// TwinCAT 3 PLC project SPS1
// Title: SPS PlattformCD
// Company: Gesim
// Author: U.Seifert
// ProjectVersion: 2.0.18.17
// ProgramVersion: 3.1.4022.4
// CompilerDefines: C6015, WIN10
// libraries:
//   Tc2_Math, * (Beckhoff Automation GmbH)
//   Tc2_NCI, * (Beckhoff Automation GmbH)
//   Tc2_Standard, * (Beckhoff Automation GmbH)
//   Tc2_System, * (Beckhoff Automation GmbH)
//   Tc3_Interfaces, * (Beckhoff Automation GmbH)
//   Tc3_Module, * (Beckhoff Automation GmbH)
//   Tc3_PackML, * (Beckhoff Automation GmbH)
//   Tc2_EtherCAT,newest,Beckhoff Automation GmbH
//   Tc2_IoFunctions,newest,Beckhoff Automation GmbH
//   Tc2_MC2,newest,Beckhoff Automation GmbH
//   Tc2_SerialCom,newest,Beckhoff Automation GmbH
//   Tc2_SUPS,newest,Beckhoff Automation GmbH
//   Tc2_SystemCX,newest,Beckhoff Automation GmbH
//   Tc2_Utilities,newest,Beckhoff Automation GmbH
//   Tc3_LinMot,1.0.0.3,NTI AG
//   Tc3_MemMan,newest,Beckhoff Automation GmbH
// project tree:
//   Actions/ ActionDispacher.TcPOU, FB_ActionList.TcPOU, FB_ActionStatusList.TcPOU, FB_ComplexAction.TcPOU, FB_DelayAction.TcPOU, FB_MeasTip.TcPOU, FB_MoveToTarget.TcPOU
//   / ComTask.TcTTO, GCodeTask.TcTTO, PlcTask.TcTTO
//   Configuration/ FB_Configuration.TcPOU, FB_GetObjPropChecksum.TcPOU, FB_IdPool.TcPOU, FB_ObjCollection.TcPOU, FB_ObjCollectionNode.TcPOU, FB_ObjCollectIterator.TcPOU, FB_ObjCollectIteratorDeep.TcPOU, FB_ObjectDirectory.TcPOU, GVL_ObjectArrays.TcGVL, GVL_ObjectConstants.TcGVL, GVL_ObjMgmt.TcGVL, ST_IdNode.TcDUT
//   DUTs/Enums/ E_ActionStatus.TcDUT, E_ArrayOrder.TcDUT, E_Condition.TcDUT, E_CrashAvoidanceMode.TcDUT, E_DilPrepareMode.TcDUT, E_DilPumpMode.TcDUT, E_DilType.TcDUT, E_DilValveType.TcDUT, E_DispenserState.TcDUT, E_DrivingPinCtrl.TcDUT, E_DrivingPinSelection.TcDUT, E_DrivingPinState.TcDUT, E_ErrorIdDS402.TcDUT, E_ErrorIdGCode.TcDUT, E_ErrorIdCan.TcDUT, E_ErrorIdHwGeneral.TcDUT, E_ExchangePieceOption.TcDUT, E_ExtruderType.TcDUT, E_GCodeState.TcDUT, E_GripperState.TcDUT, E_HardwarePropType.TcDUT, E_InteractMessageType.TcDUT, E_InterlockState.TcDUT, E_CompOperator.TcDUT, E_LockCtrl.TcDUT, E_LockState.TcDUT, E_MeasureMode.TcDUT, E_MeasureOption.TcDUT, E_MethodState.TcDUT, E_ModalDesignationAbsInc.TcDUT, E_ModalGeoTypes.TcDUT, E_MoveDirection.TcDUT, E_MoveMode.TcDUT, E_ObjectGroup.TcDUT, E_OpClCtrl.TcDUT, E_OpClState.TcDUT, E_LogicOperator.TcDUT, E_PickPutMode.TcDUT, E_POU.TcDUT, E_POUACT.TcDUT, E_PressCtrl.TcDUT, E_PrintParamType.TcDUT, E_ProcDataType.TcDUT, E_StackerRotPosition.TcDUT, E_SwivelCtrl.TcDUT, E_SwivelState.TcDUT, E_TargetRef.TcDUT, E_Action.TcDUT, E_ErrorIdCmd.TcDUT, E_ErrorIdDiluter.TcDUT, E_ErrorIdMultiZ.TcDUT, E_HardwareGrp.TcDUT, E_MachineMode.TcDUT, E_MachineState.TcDUT, E_ObjectType.TcDUT, E_ErrorIdObjMgmt.TcDUT, E_TeachTrgtOption.TcDUT, E_TipCleaningMode.TcDUT, E_TransferTrayCtrl.TcDUT, E_TrayHollowSelection.TcDUT, E_TriggerOutput.TcDUT, E_WashMode.TcDUT
//   DUTs/ ERRORID.TcDUT, HARDWAREGRP.TcDUT
//   DUTs/Structs/ FB_Rectangle.TcPOU, ST_Action.TcDUT, ST_ActionStatus.TcDUT, ST_2DPoint.TcDUT, ST_3DDimension.TcDUT, ST_3DPoint.TcDUT, ST_ActionData.TcDUT, ST_ActionList.TcDUT, ST_AdsAdress.TcDUT, ST_CanMasterAddress.TcDUT, ST_Circle.TcDUT, ST_EtherCATMaster.TcDUT, ST_HardwareProcData.TcDUT, ST_HardwareId.TcDUT, ST_HardwareInfo.TcDUT, ST_Interaction.TcDUT, ST_Line.TcDUT, ST_MethResult.TcDUT, ST_ObjHasMoved.TcDUT, ST_PlcInfo.TcDUT, ST_ObjectProcData.TcDUT, ST_Rectangle.TcDUT, ST_CmdData.TcDUT, ST_Error.TcDUT, ST_StepStatus.TcDUT, ST_WashPoint.TcDUT, ST_WashStep.TcDUT, ST_WasteChannel.TcDUT, ST_LiquidChannel.TcDUT, ST_RinseChannel.TcDUT
//   DUTs/Unions/ U_AdsData.TcDUT, U_ByteArr4_DINT.TcDUT, U_SDO_DATA.TcDUT
//   FirmwUpdate/ E_FirmwUpdState.TcDUT, E_S19RecordState.TcDUT, FB_S19File.TcPOU, FB_S19Record.TcPOU, FirmwUpdate.TcPOU, ST_FirmwUpdInfo.TcDUT
//   Functions/ F_Add3DPoints.TcPOU, F_CuboidInnerCuboid.TcPOU, F_GET_GCODE_NCLINE.TcPOU, F_Sub3DPoints.TcPOU, F_SynchronizeSpeeds.TcPOU
//   GCode/ E_SAF_State.TcDUT, FB_BuildGroup.TcPOU, FB_ClearGroup.TcPOU, FB_Cuboid.TcPOU, FB_FastMFunc.TcPOU, FB_HskMFunc.TcPOU, FB_RestartPrintAction.TcPOU, GCode.TcPOU, ST_GCodeInfo2.TcDUT, ST_GCodeRef.TcDUT, ST_GCodeTool.TcDUT, ST_NciInfo.TcDUT, ST_GCodeInfo.TcDUT
//   GVLs/ GVL_Hardware.TcGVL, GVL_RS232.TcGVL, GVL_Sm.TcGVL
//   Hardware/4ChannelHeater/ FB_HwRef4ChHeater.TcPOU
//   Hardware/BottleRack/ FB_HwRefBottleRack.TcPOU
//   Hardware/ CANInterfaceCom.TcPOU, E_CoDS402HomingState.TcDUT, E_CoDS402States.TcDUT, FB_CanNodeBase.TcPOU, FB_CANOpenMotionPower.TcPOU, FB_HwModule.TcPOU, FB_HwModuleList.TcPOU, FB_SendCanMessage.TcPOU, F_GetCoDS402State.TcPOU, F_CompVersion.TcPOU, HwInfoList.TcPOU, PerformHardware.TcPOU, ScanHwModules.TcPOU, SimutateHwModules.TcPOU, ST_CANInterfaceBuffer.TcDUT
//   Hardware/Diluter/ FB_Dil_GetValveConfig.TcPOU, FB_Dil_GetValvePos.TcPOU, FB_Dil_GetPlungerPos.TcPOU, FB_Dil_Pump.TcPOU, FB_Dil_MoveValve.TcPOU, FB_Dil_MoveToPos.TcPOU, FB_Dil_SendCmd.TcPOU, FB_Dil_SetValveConfig.TcPOU, FB_Dil_Transfer.TcPOU, FB_Dil_Init.TcPOU, FB_Dil_Stop.TcPOU, FB_HwRefDiluter.TcPOU, F_DilFlowToSpeed.TcPOU, F_DilQuantityToMicroSteps.TcPOU, F_GetChannelCodeTwin.TcPOU, F_GetCheckSumByte.TcPOU, F_GetCheckSumFromString.TcPOU, F_GetPumpString.TcPOU, F_GetValveCode.TcPOU
//   Hardware/EL70xxDrive/ E_EL70xx_EncoderType.TcDUT, E_EL70xx_StartType.TcDUT, FB_HWECtrl_EL70xx_Home.TcPOU, FB_HWECtrl_EL70xx_Move.TcPOU, FB_HWECtrl_EL70xx_Power.TcPOU, FB_HwRefEL70xxDrive.TcPOU, FB_HwRefEL70xxDriveExtEncoder.TcPOU, ST_EL70xx_POS_Control.TcDUT, ST_EL70xx_POS_Status.TcDUT, ST_EL70xx_STM_Control.TcDUT, ST_EL70xx_STM_Status.TcDUT
//   Hardware/FBox/ FB_HwRefMultiPurpIO.TcPOU, FB_PCV.TcPOU, FB_Pump.TcPOU, FB_HwRefTripleTrigger.TcPOU, FB_Valve.TcPOU, F_YFuncX.TcPOU
//   Hardware/FBox/PneuChannels/ FB_PneuChannelRef.TcPOU, FB_SetPressure.TcPOU
//   Hardware/HuberUnistat/ E_UnistatState.TcDUT, E_Unitstat_Command.TcDUT, FB_HwRefUnistat.TcPOU, FB_UnistatControl.TcPOU, FB_Unistat_SendCmd.TcPOU
//   Hardware/IOExpander/ FB_PulseTrainControl.TcPOU, ST_PulseTrainChannel.TcDUT, FB_HwRefIOExpander.TcPOU
//   Hardware/MultiZ/Extruder/ FB_EndlessExtruderTMCM_Control.TcPOU, FB_EndlessExtruderTMCM_Ref.TcPOU, FB_FDM_EL2521_Control.TcPOU, FB_FDM_EL2521_Ref.TcPOU, FB_ExtruderControl.TcPOU, FB_ExtruderRef.TcPOU, FB_PistonExtruderControl.TcPOU, FB_PistonExtruderRef.TcPOU
//   Hardware/MultiZ/Gripper/ FB_GripperRef.TcPOU
//   Hardware/MultiZ/Heater/ E_MzHeaterType.TcDUT, FB_MzHeaterControl.TcPOU, FB_MZHeaterRef.TcPOU
//   Hardware/MultiZ/PWM/ FB_MultiZPWM.TcPOU
//   Hardware/NanotecPanDrive/ FB_HwRefNanotecPD.TcPOU, FB_NanotecPD_Home.TcPOU, FB_NanotecPD_Move.TcPOU, FB_NanotecPD_Power.TcPOU
//   Hardware/RS232/ FB_SerialComPort_Base.TcPOU, FB_SerialComPort_EL60xx.TcPOU, FB_SerialComPort_PC.TcPOU, FB_SerialComPort_USB.TcPOU, FB_SimpleFIFO_PVOID.TcPOU, SerialBackCom.TcPOU
//   Hardware/Safety/ E_SafetyCtrl.TcDUT, E_SafetyState.TcDUT, FB_Safety.TcPOU, FB_SafetyPseudo.TcPOU, FB_SafetyBase.TcPOU, FB_HwRefStopButton.TcPOU, FB_SafetyStacker.TcPOU, FB_SignalLight.TcPOU
//   Hardware/HighVoltSupply/ FB_HighVoltSupply.TcPOU
//   Hardware/InkStation/ FB_HwRefInkStatDriveCover.TcPOU, FB_HwRefInkStatDriveSpin.TcPOU, FB_InkStationInitSpinDrive.TcPOU, FB_InkStationInitCoverDrive.TcPOU, FB_InkStationOpenClose.TcPOU
//   Hardware/LiquidReserve/ E_TMCMCommand.TcDUT, FB_GearPump.TcPOU, FB_TMCM6110.TcPOU
//   Hardware/MultiZ/ E_MzToolType.TcDUT, FB_MultiZRef.TcPOU, FB_MultiZStamp.TcPOU, FB_MultiZTipEjector.TcPOU, FB_ZAxisRef.TcPOU, FB_ZM_Home.TcPOU, FB_ZM_Jog.TcPOU, FB_ZM_Move.TcPOU, FB_ZM_ReadZSensorID.TcPOU, FB_ZM_Stop.TcPOU, F_MultiZError_TO_ErrorId.TcPOU, GVL_MultiZObjects.TcGVL, ST_CANopenObject.TcDUT, ST_StampSupport.TcDUT, ST_StrobTrigger.TcDUT, ST_ZAxisRef_In.TcDUT, ST_ZAxisRef_Out.TcDUT, ST_ZAxisStatus.TcDUT, ST_ZGPIO_AnaIn.TcDUT, ST_ZGPIO_PWM_ANA.TcDUT, ST_ZSensorCalibration.TcDUT
//   Hardware/MultiZ/GPIO/ E_GPInputMode.TcDUT, FB_GPInputRef.TcPOU
//   Hardware/MultiZ/Piezo/ E_DispenserMode.TcDUT, FB_PiezoControl.TcPOU, FB_PiezoRef.TcPOU
//   Hardware/PTOStepper/ FB_PTOStepperMoveRel.TcPOU, FB_PTOStepperRotate.TcPOU, ST_PTOStepperRef.TcDUT
//   Hardware/PowderStation/ FB_HwRefPowderStat.TcPOU
//   Hardware/Reactor/ E_ReactDrive.TcDUT, FB_ReactDriveInit.TcPOU, FB_ReactDriveMove.TcPOU, FB_HwRefReactDrive.TcPOU, FB_HwRefReactHeater.TcPOU
//   Hardware/SDO_Com/ FB_SDO_READ.TcPOU, FB_SDO_WRITE.TcPOU, F_AdsError_TO_SdoError.TcPOU
//   Hardware/Settings/ FB_Settings.TcPOU
//   Hardware/TipCalibrator/ ST_TipCalibrator.TcDUT
//   Hardware/TipCleaner/ FB_TipCleanerInit.TcPOU, ST_TipCleanerRef.TcDUT
//   Hardware/TMCM-1140/ E_TMCM_HomingMethode.TcDUT, E_TMCM_SwitchConfig.TcDUT, E_TMCM_VeloDim.TcDUT, FB_HwRefTMCM1140.TcPOU, FB_TMCM1140_Home.TcPOU, FB_TMCM1140_Move.TcPOU, FB_TMCM1140_Power.TcPOU, FB_TMCM1140_Rotate.TcPOU
//   Hardware/TrayLock/ FB_HwRefTrayLock.TcPOU, FB_HwTrayLockControl.TcPOU
//   Hardware/Trigger/ FB_TriggerOut.TcPOU, GVL_HwRefIO.TcGVL, OutDistributor.TcPOU
//   Hardware/XYDrive/ CoupleYY.TcPOU, E_XYOrientation.TcDUT, FB_LmtChangePID.TcPOU, FB_XYDriveBase.TcPOU, FB_XYDriveNC.TcPOU, FB_XYDrive_Beck_Twin.TcPOU, FB_XYDrive_Beck.TcPOU, FB_XYDrive_Lmt_DS.TcPOU, FB_XYDrive_Lmt_EC.TcPOU
//   MainProgs/ MainDispacher.TcPOU, PC_Control.TcPOU, MAIN.TcPOU
//   Objects/Devices/ FB_Diluter3Inputs.TcPOU, FB_Diluter.TcPOU, FB_Stacker.TcPOU
//   Objects/ FB_DimSlot.TcPOU, FB_Object.TcPOU, FB_PieceSlot.TcPOU, FB_Slot.TcPOU, FB_SlotList.TcPOU, F_GetTwoLineAngle.TcPOU, F_LinesIntersect.TcPOU, F_PointInnerRect.TcPOU, F_RectInnerCircle.TcPOU, F_RectInnerRect.TcPOU, F_RectIntersectRect.TcPOU, F_RotatePoint.TcPOU, ST_Shelf.TcDUT, ST_POINTER2.TcDUT
//   Objects/Interfaces/ I_Dispenser.TcIO, I_SlotTarget.TcIO, I_Device.TcIO, I_TargetZSensor.TcIO, I_UsingDryPad.TcIO
//   Objects/Pieces/ FB_Cartridge.TcPOU, FB_Needle.TcPOU, FB_Nozzle.TcPOU, FB_pHElectrodeCap.TcPOU, FB_PieceBase.TcPOU, FB_Port.TcPOU, FB_Tip.TcPOU, FB_VialClosed.TcPOU, FB_FlipTube.TcPOU, FB_Stamp.TcPOU, FB_Septum.TcPOU, FB_UsingPiece.TcPOU, FB_Vial.TcPOU
//   Objects/Targets/Active/ FB_ActiveTarget.TcPOU, FB_CustomUnitType1.TcPOU, FB_CustomUnitType2.TcPOU, FB_HighVoltTray.TcPOU, FB_InkStation.TcPOU, FB_LiquidReserve.TcPOU, FB_MtpHolder.TcPOU, FB_PowderStation.TcPOU, FB_Reactor.TcPOU, FB_Stroboscope.TcPOU, FB_SubstHolder.TcPOU, FB_SubstHolderUnistat.TcPOU, FB_TipCalibrator.TcPOU, FB_TipCleaner.TcPOU, FB_TrayTransporter.TcPOU, FB_WashStation.TcPOU, FB_WorkplateCamera.TcPOU
//   Objects/Targets/ FB_TargetBase.TcPOU
//   Objects/Targets/Passive/ FB_Array.TcPOU, FB_CleaningBrush.TcPOU, FB_DryPad.TcPOU, FB_FlipTubeRack.TcPOU, FB_Mtp.TcPOU, FB_NeedleRack.TcPOU, FB_pHElectrodeCapRack.TcPOU, FB_Point.TcPOU, FB_PortRack.TcPOU, FB_Rack.TcPOU, FB_SeptumRack.TcPOU, FB_SeptumWaste.TcPOU, FB_Slide.TcPOU, FB_SlotTarget.TcPOU, FB_SpotArray.TcPOU, FB_SpotPattern.TcPOU, FB_StampMagazine.TcPOU, FB_TargetTray.TcPOU, FB_TipCleanerGen2.TcPOU, FB_TipRack.TcPOU, FB_VialRack.TcPOU, FB_Wafer.TcPOU, FB_Workplate.TcPOU
//   Objects/Tools/ FB_Camera.TcPOU, FB_CartDispenser.TcPOU, FB_CartDispStirrer.TcPOU, FB_CartHolder.TcPOU, FB_DummyTool.TcPOU, FB_Extruder.TcPOU, FB_DeloDot.TcPOU, FB_Exposure.TcPOU, FB_FlipTubeHandler.TcPOU, FB_GCodeTool.TcPOU, FB_Gripper.TcPOU, FB_HybridDispenser.TcPOU, FB_MultiCartHolder.TcPOU, FB_pHElectrode.TcPOU, FB_PickPlacePip.TcPOU, FB_SingelPiezoHolder.TcPOU, FB_SolenoidPip.TcPOU, FB_TitrationTool.TcPOU, FB_TwinExtruder.TcPOU, FB_TwinPiezoHolder.TcPOU, FB_MzBase.TcPOU, FB_MzHead.TcPOU, FB_MzTool.TcPOU, FB_PassivPip.TcPOU, FB_Luer.TcPOU, FB_TriplePip.TcPOU, FB_PiezoPip.TcPOU, FB_PowderPip.TcPOU, FB_StampSupport.TcPOU, FB_VacuumHandler.TcPOU, FB_VermesDisp.TcPOU, FB_ZLevelSensor.TcPOU
//   Error/ FB_ErrorList.TcPOU
//   Sequence/ E_SequenceState.TcDUT, E_StepState.TcDUT, FB_CondiBase.TcPOU, FB_CondiStepResult.TcPOU, FB_CondiStepReady.TcPOU, FB_CondiProcessData.TcPOU, FB_ProcessingQueue.TcPOU, FB_SequenceInfo.TcPOU, FB_SequenceList.TcPOU, FB_StepList.TcPOU, FB_Sequence.TcPOU, F_SetFollowerStep.TcPOU, ST_Pointer.TcDUT, ST_SequenceInfo.TcDUT, ST_Step.TcDUT
//   OperatingModes/ FB_OM_Auto.TcPOU, FB_OM_Config.TcPOU, FB_OM_Init.TcPOU, FB_OM_Maintenance.TcPOU, FB_OM_Manu.TcPOU, FB_OM_SemiAuto.TcPOU
//   Version/ Global_Version.TcGVL
// real-time tasks:
//   TASK ComTask: cycle T#4ms, priority 8, ADS port 350
//   TASK GCodeTask: cycle T#2ms, priority 6, ADS port 351
//   TASK PlcTask: cycle T#10ms, priority 14, ADS port 352
// motion (NC):
//   TASK NC-Task 1 SAF: cycle T#2ms, priority 4, ADS port 501
//   TASK NC-Task 1 SVB: cycle T#10ms, priority 12, ADS port 511
//   AXIS Achse 1 (X) (id 1)
//     Dynamic: AccelerationMaximum=20000, DecelerationMaximum=20000, Acceleration=1533.33, Deceleration=1533.33, Jerk=20444.4
//     Velo: Fast=20, Maximum=150
//     OtherSettings: AllowMotionCmdToSlave=true
//     encoder EncType=19
//       EncPara: Inverse=true, MaxCount=#xffffffff
//     drive DrvType=16
//       DrvPara: Inverse=true, MaxCount=#xffffffff
//         Analog: ScaleFactorActTorque=0.1
//         TimeComp: TaskDelayCycles=1
//     controller CtrType=1
//       CtrPara: PriorControlFactor=1
//         PID: CtrlOutputLimit=0
//         Observer: BandWidth=20
//   AXIS Achse 2 (Y) (id 2)
//     Dynamic: AccelerationMaximum=20000, DecelerationMaximum=20000, Acceleration=1502.67, Deceleration=1502.67, Jerk=20453
//     Velo: Fast=20, Maximum=150
//     OtherSettings: AllowMotionCmdToSlave=true
//     encoder EncType=19
//       EncPara: MaxCount=#xffffffff
//         SoftEndMaxControl: Range=330
//     drive DrvType=16
//       DrvPara: MaxCount=#xffffffff
//         Analog: ScaleFactorActTorque=0.1
//         TimeComp: TaskDelayCycles=1
//     controller CtrType=1
//       CtrPara: PriorControlFactor=1
//         PID: CtrlOutputLimit=0
//         Observer: BandWidth=20
//   AXIS Achse 4 Q1 (id 4)
//     General: UnitName=
//     OtherSettings: AllowMotionCmdToSlave=true
//     encoder EncType=1
//     drive DrvType=5
//       TimeComp: TaskDelayCycles=1
//     controller CtrType=1
//       CtrPara: PriorControlFactor=1
//         Observer: BandWidth=20
// I/O:
//   DEVICE Gerät 1 (EL6751), AmsNetId 192.168.135.178.2.1
//     CAN Interface
//     CAN 1 (TraySlider Nanotec PD2-C) (disabled)
//     CAN 8 (MultiZ 1)
//     CAN 10(MtpHeater1) (disabled)
//     CAN12(SubstHeater1) (disabled)
//     CAN 35 (TMCM-Driving pin right) (disabled)
//     CAN 36 (TMCM-Driving pin left) (disabled)
//     CAN25 (MultiPurpIO)
//   DEVICE Gerät 3 (EtherCAT), AmsNetId 192.168.135.178.4.1
//     -KL01 (EK1100) [EK1100 EtherCAT-Koppler (2A E-Bus)]
//       -KL07 (EL1918) [EL1918, 8K. Safety Eingang 24V, TwinSAFE]
//         modules: Module 2 (FSLOGIC)
//       -KL08 (EL2904) [EL2904, 4 K. Safety Ausgang 24V, 0.5A, TwinSAFE]
//         modules: Module 1 (FSOES), Module 2 (DO)
//       -KL10 (EL6751) [EL6751 CANopen Master]
//       End(EL9011) [EL9011 Endklemme]
//     Drive1 (C1250-DS-XC-1S)X [C1250-DS-XC-1S V1.8b5]
//     Drive2 (C1250-DS-XC-1S)Y [C1250-DS-XC-1S V1.8b5]
// variable links:
//   Device 3 (EtherCAT) <-> Device 3 (EtherCAT)/-KL01 (EK1100)/-KL07 (EL1918)
//     -KL01 (EK1100)/-KL08 (EL2904)/Module 1 (FSOES)/RxPDO/FSOE <-> ConnectionInputs/Message_22 TxPDO
//     -KL01 (EK1100)/-KL08 (EL2904)/Module 1 (FSOES)/TxPDO/FSOE <-> ConnectionOutputs/Message_22 RxPDO
//   NC-Task 1 SAF/Axes/Achse 1 (X) <-> Device 3 (EtherCAT)/Drive1 (C1250-DS-XC-1S)X
//     Drive/Inputs/In/nDcOutputTime <-> InfoData/DcOutputShift
//     Drive/Inputs/In/nState1 <-> Cylic Mode Inputs/Statusword
//     Drive/Inputs/In/nState2 <-> Cylic Mode Inputs/Statusword @bit 8
//     Drive/Inputs/In/nState4 @bit 1 <-> WcState/InputToggle
//     Drive/Inputs/In/nState4 <-> WcState/WcState
//     Drive/Inputs/In/nState5 <-> Cylic Mode Inputs/Mode of Operation display
//     Drive/Outputs/Out/nCtrl1 <-> Cylic Position Velocity Mode/Controlword
//     Drive/Outputs/Out/nCtrl2 <-> Cylic Position Velocity Mode/Controlword @bit 8
//     Drive/Outputs/Out/nCtrl5 <-> Cylic Position Velocity Mode/Mode of Operation
//     Drive/Outputs/Out/nDataOut1 <-> Cylic Position Velocity Mode/Target position
//     Drive/Outputs/Out/nDataOut2 <-> Cylic Position Velocity Mode/Target velocity
//     Enc/Inputs/In/nDataIn1 <-> Cylic Mode Inputs/Position actual value (units)
//     Enc/Inputs/In/nDcInputTime <-> InfoData/DcInputShift
//     Enc/Inputs/In/nState4 @bit 1 <-> WcState/InputToggle
//     Enc/Inputs/In/nState4 <-> WcState/WcState
//   NC-Task 1 SAF/Axes/Achse 2 (Y) <-> Device 3 (EtherCAT)/Drive2 (C1250-DS-XC-1S)Y
//     Drive/Inputs/In/nDcOutputTime <-> InfoData/DcOutputShift
//     Drive/Inputs/In/nState1 <-> Cylic Mode Inputs/Statusword
//     Drive/Inputs/In/nState2 <-> Cylic Mode Inputs/Statusword @bit 8
//     Drive/Inputs/In/nState4 @bit 1 <-> WcState/InputToggle
//     Drive/Inputs/In/nState4 <-> WcState/WcState
//     Drive/Inputs/In/nState5 <-> Cylic Mode Inputs/Mode of Operation display
//     Drive/Outputs/Out/nCtrl1 <-> Cylic Position Velocity Mode/Controlword
//     Drive/Outputs/Out/nCtrl2 <-> Cylic Position Velocity Mode/Controlword @bit 8
//     Drive/Outputs/Out/nCtrl5 <-> Cylic Position Velocity Mode/Mode of Operation
//     Drive/Outputs/Out/nDataOut1 <-> Cylic Position Velocity Mode/Target position
//     Drive/Outputs/Out/nDataOut2 <-> Cylic Position Velocity Mode/Target velocity
//     Enc/Inputs/In/nDataIn1 <-> Cylic Mode Inputs/Position actual value (units)
//     Enc/Inputs/In/nDcInputTime <-> InfoData/DcInputShift
//     Enc/Inputs/In/nState4 @bit 1 <-> WcState/InputToggle
//     Enc/Inputs/In/nState4 <-> WcState/WcState
//   SPS1/SPS1 Instance <-> Device 1 (EL6751)/CAN 10(MtpHeater1)
//     PlcTask Inputs/GVL_Hardware.aFbMtpHeatRef[1].bTempCutoff <-> TxPDO 1/Inputs/TempCutoff
//     PlcTask Inputs/GVL_Hardware.aFbMtpHeatRef[1].nNodeState <-> Inputs/NodeState
//     PlcTask Inputs/GVL_Hardware.aFbMtpHeatRef[1].nTempActual <-> TxPDO 1/Inputs/TempActual
//     PlcTask Outputs/GVL_Hardware.aFbMtpHeatRef[1].bEdgeLightOn <-> RxPDO 2/Outputs/EdgeLightOn
//     PlcTask Outputs/GVL_Hardware.aFbMtpHeatRef[1].bHeatingOn <-> RxPDO 2/Outputs/HeatingOn
//     PlcTask Outputs/GVL_Hardware.aFbMtpHeatRef[1].nPidKd <-> RxPDO 1/Outputs/PID_Kd
//     PlcTask Outputs/GVL_Hardware.aFbMtpHeatRef[1].nPidKi <-> RxPDO 1/Outputs/PID_Ki
//     PlcTask Outputs/GVL_Hardware.aFbMtpHeatRef[1].nPidKp <-> RxPDO 1/Outputs/PID_Kp
//     PlcTask Outputs/GVL_Hardware.aFbMtpHeatRef[1].nPidTa <-> RxPDO 1/Outputs/PID_Ta
//     PlcTask Outputs/GVL_Hardware.aFbMtpHeatRef[1].nTempSetpoint <-> RxPDO 2/Outputs/TempSetpoint
//   SPS1/SPS1 Instance <-> Device 1 (EL6751)/CAN 8 (MultiZ 1)
//     PlcTask Inputs/GVL_Hardware.aFbMultiZRef[1].aFbExtruderRef[1].nCurrentPlungerPos <-> TxPDO 11/Inputs/HT-Extrud-CurrPos-Z12
//     PlcTask Inputs/GVL_Hardware.aFbMultiZRef[1].aFbExtruderRef[2].nCurrentPlungerPos <-> TxPDO 11/Inputs/HT-Extrud-CurrPos-Z12
//     PlcTask Inputs/GVL_Hardware.aFbMultiZRef[1].aFbExtruderRef[3].nCurrentPlungerPos <-> TxPDO 11/Inputs/HT-Extrud-CurrPos-Z34
//     PlcTask Inputs/GVL_Hardware.aFbMultiZRef[1].aFbExtruderRef[4].nCurrentPlungerPos <-> TxPDO 11/Inputs/HT-Extrud-CurrPos-Z34
//     PlcTask Inputs/GVL_Hardware.aFbMultiZRef[1].aFbExtruderRef[5].nCurrentPlungerPos <-> TxPDO 12/Inputs/HT-Extrud-CurrPos-Z56
//     PlcTask Inputs/GVL_Hardware.aFbMultiZRef[1].aFbExtruderRef[6].nCurrentPlungerPos <-> TxPDO 12/Inputs/HT-Extrud-CurrPos-Z56
//     PlcTask Inputs/GVL_Hardware.aFbMultiZRef[1].aFbExtruderRef[7].nCurrentPlungerPos <-> TxPDO 12/Inputs/HT-Extrud-CurrPos-Z7
//     PlcTask Inputs/GVL_Hardware.aFbMultiZRef[1].aFbGPInputRef[1].nValue <-> TxPDO 14/Inputs/Ana/Digi-Input-Value-Z1
//     PlcTask Inputs/GVL_Hardware.aFbMultiZRef[1].aFbGPInputRef[2].nValue <-> TxPDO 14/Inputs/Ana/Digi-Input-Value-Z2
//     PlcTask Inputs/GVL_Hardware.aFbMultiZRef[1].aFbGPInputRef[3].nValue <-> TxPDO 14/Inputs/Ana/Digi-Input-Value-Z3
//     PlcTask Inputs/GVL_Hardware.aFbMultiZRef[1].aFbGPInputRef[4].nValue <-> TxPDO 14/Inputs/Ana/Digi-Input-Value-Z4
//     PlcTask Inputs/GVL_Hardware.aFbMultiZRef[1].aFbGPInputRef[5].nValue <-> TxPDO 15/Inputs/Ana/Digi-Input-Value-Z5
//     PlcTask Inputs/GVL_Hardware.aFbMultiZRef[1].aFbGPInputRef[6].nValue <-> TxPDO 15/Inputs/Ana/Digi-Input-Value-Z6
//     PlcTask Inputs/GVL_Hardware.aFbMultiZRef[1].aFbHeaterRef[{1..7}].bHeaterIsOn <-> TxPDO 10/Inputs/Tool-State-Z{1..7} @bit 2  (7 links)
//     PlcTask Inputs/GVL_Hardware.aFbMultiZRef[1].aFbHeaterRef[{1..7}].nTemp1Actual <-> TxPDO {3..9}/Inputs/TempActual-Z{1..7}  (7 links)
//     PlcTask Inputs/GVL_Hardware.aFbMultiZRef[1].aFbHeaterRef[{1..7}].nTemp2Actual <-> TxPDO {3..9}/Inputs/TempActual2-Z{1..7}  (7 links)
//     PlcTask Inputs/GVL_Hardware.aFbMultiZRef[1].aFbZAxisRef[{1..7}].stInput.nCurrentPos <-> TxPDO {3..9}/Inputs/Current-Position-Z{1..7}  (7 links)
//     PlcTask Inputs/GVL_Hardware.aFbMultiZRef[1].aFbZAxisRef[{1..7}].stInput.nError <-> TxPDO 2/Inputs/Error-Z{1..7}  (7 links)
//     PlcTask Inputs/GVL_Hardware.aFbMultiZRef[1].aFbZAxisRef[{1..7}].stInput.nStatus <-> TxPDO 1/Inputs/Status-Byte-Z{1..7}  (7 links)
//     PlcTask Inputs/GVL_Hardware.aFbMultiZRef[1].aFbZAxisRef[{1..7}].stInput.nToolState <-> TxPDO 10/Inputs/Tool-State-Z{1..7}  (7 links)
//     PlcTask Inputs/GVL_Hardware.aFbMultiZRef[1].nErrorGlobal <-> TxPDO 2/Inputs/Error-Global
//     PlcTask Inputs/GVL_Hardware.aFbMultiZRef[1].nNodeState <-> Inputs/NodeState
//     PlcTask Inputs/GVL_Hardware.aFbMultiZRef[1].stStampSupport.bAngleReached <-> TxPDO 1/Inputs/uCP-Stamp-State
//     PlcTask Inputs/GVL_Hardware.aFbMultiZRef[1].stStampSupport.bError <-> TxPDO 1/Inputs/uCP-Stamp-State @bit 4
//     PlcTask Inputs/GVL_Hardware.aFbMultiZRef[1].stStampSupport.bInitLockOk <-> TxPDO 1/Inputs/uCP-Stamp-State @bit 3
//     PlcTask Inputs/GVL_Hardware.aFbMultiZRef[1].stStampSupport.bInitSpinOk <-> TxPDO 1/Inputs/uCP-Stamp-State @bit 2
//     PlcTask Inputs/GVL_Hardware.aFbMultiZRef[1].stStampSupport.bLocked <-> TxPDO 1/Inputs/uCP-Stamp-State @bit 1
//     PlcTask Inputs/GVL_Hardware.aFbMultiZRef[1].stStampSupport.bStampInMagazine <-> TxPDO 1/Inputs/uCP-Stamp-State @bit 5
//     PlcTask Inputs/GVL_Hardware.aFbMultiZRef[1].stStampSupport.bStampInSupport <-> TxPDO 1/Inputs/uCP-Stamp-State @bit 6
//     PlcTask Outputs/GVL_Hardware.aFbMultiZRef[1].aDigiOut[5] <-> RxPDO 11/Outputs/Digital-Output-Z5
//     PlcTask Outputs/GVL_Hardware.aFbMultiZRef[1].aDigiOut[6] <-> RxPDO 11/Outputs/Digital-Output-Z6
//     PlcTask Outputs/GVL_Hardware.aFbMultiZRef[1].aDigiOut[7] <-> RxPDO 11/Outputs/Digital-Output-Z7
//     PlcTask Outputs/GVL_Hardware.aFbMultiZRef[1].aFbZAxisRef[{1..7}].stOutput.nCtrl <-> RxPDO 1/Outputs/Control-Byte-Z{1..7}  (7 links)
//     PlcTask Outputs/GVL_Hardware.aFbMultiZRef[1].aFbZAxisRef[{1..7}].stOutput.nMode <-> RxPDO 2/Outputs/Operation-Mode-Z{1..7}  (7 links)
//     PlcTask Outputs/GVL_Hardware.aFbMultiZRef[1].aFbZAxisRef[{1..7}].stOutput.nToolCtrl <-> RxPDO 10/Outputs/Tool-Ctrl-Z{1..7}  (7 links)
//     PlcTask Outputs/GVL_Hardware.aFbMultiZRef[1].aFbZAxisRef[{1..7}].stOutput.nTrgtPos <-> RxPDO {3..9}/Outputs/Target-Position-Z{1..7}  (7 links)
//     PlcTask Outputs/GVL_Hardware.aFbMultiZRef[1].aFbZAxisRef[{1..7}].stOutput.nVelo <-> RxPDO {3..9}/Outputs/Velocity-Z{1..7}  (7 links)
//     PlcTask Outputs/GVL_Hardware.fbMultiZDigiOut.aOut[1] <-> RxPDO 11/Outputs/Digital-Output-Z2
//     PlcTask Outputs/GVL_Hardware.fbMultiZDigiOut.aOut[2] <-> RxPDO 11/Outputs/Digital-Output-Z3
//     PlcTask Outputs/GVL_Hardware.fbMultiZDigiOut.aOut[3] <-> RxPDO 11/Outputs/Digital-Output-Z4
//     PlcTask Outputs/GVL_Hardware.fbMultiZPWM.aEnable[1] <-> RxPDO 12/Outputs/PWM1_Enable
//     PlcTask Outputs/GVL_Hardware.fbMultiZPWM.aEnable[2] <-> RxPDO 12/Outputs/PWM2_Enable
//     PlcTask Outputs/GVL_Hardware.fbMultiZPWM.aValue[1] <-> RxPDO 12/Outputs/PWM1_Value
//     PlcTask Outputs/GVL_Hardware.fbMultiZPWM.aValue[2] <-> RxPDO 12/Outputs/PWM2_Value
//   SPS1/SPS1 Instance <-> Device 1 (EL6751)/CAN Interface
//     ComTask Inputs/CANInterfaceCom.aInData <-> Inputs/RxQueue/RxMessages[0]/data
//     ComTask Inputs/CANInterfaceCom.nInCobId <-> Inputs/RxQueue/RxMessages[0]/cobId
//     ComTask Inputs/CANInterfaceCom.nInRxCounter <-> Inputs/RxQueue/RxCounter
//     ComTask Inputs/CANInterfaceCom.nInTxCounter <-> Inputs/RxQueue/TxCounter
//     ComTask Outputs/CANInterfaceCom.aOutData <-> Outputs/TxQueue/TxMessages[0]/data
//     ComTask Outputs/CANInterfaceCom.nOutCobId <-> Outputs/TxQueue/TxMessages[0]/cobId
//     ComTask Outputs/CANInterfaceCom.nOutNoOfTxMessages <-> Outputs/TxQueue/NoOfTxMessages
//     ComTask Outputs/CANInterfaceCom.nOutRxCounter <-> Outputs/TxQueue/RxCounter
//     ComTask Outputs/CANInterfaceCom.nOutTxCounter <-> Outputs/TxQueue/TxCounter
//   SPS1/SPS1 Instance <-> Device 1 (EL6751)/CAN12(SubstHeater1)
//     PlcTask Inputs/GVL_Hardware.aFbSubstHeatRef[1].bTempCutoff <-> TxPDO 1/Inputs/TempCutoff
//     PlcTask Inputs/GVL_Hardware.aFbSubstHeatRef[1].nNodeState <-> Inputs/NodeState
//     PlcTask Inputs/GVL_Hardware.aFbSubstHeatRef[1].nTempActual <-> TxPDO 1/Inputs/TempActual
//     PlcTask Outputs/GVL_Hardware.aFbSubstHeatRef[1].bEdgeLightOn <-> RxPDO 2/Outputs/EdgeLightOn
//     PlcTask Outputs/GVL_Hardware.aFbSubstHeatRef[1].bHeatingOn <-> RxPDO 2/Outputs/HeatingOn
//     PlcTask Outputs/GVL_Hardware.aFbSubstHeatRef[1].nPidKd <-> RxPDO 1/Outputs/PID_Kd
//     PlcTask Outputs/GVL_Hardware.aFbSubstHeatRef[1].nPidKi <-> RxPDO 1/Outputs/PID_Ki
//     PlcTask Outputs/GVL_Hardware.aFbSubstHeatRef[1].nPidKp <-> RxPDO 1/Outputs/PID_Kp
//     PlcTask Outputs/GVL_Hardware.aFbSubstHeatRef[1].nPidTa <-> RxPDO 1/Outputs/PID_Ta
//     PlcTask Outputs/GVL_Hardware.aFbSubstHeatRef[1].nTempSetpoint <-> RxPDO 2/Outputs/TempSetpoint
//   SPS1/SPS1 Instance <-> Device 1 (EL6751)/CAN25 (MultiPurpIO)
//     PlcTask Inputs/GVL_Hardware.aFbHwRefMultiPurpIO[1].nNodeState <-> Inputs/NodeState
//     PlcTask Inputs/GVL_Hardware.aFbPneuChannel[1].bSupplyOk <-> TxPDO 4/Inputs/Digi-Input-Value_5
//     PlcTask Inputs/GVL_Hardware.aFbPneuChannel[2].bSupplyOk <-> TxPDO 4/Inputs/Digi-Input-Value_5
//     PlcTask Inputs/GVL_Hardware.aFbPneuChannel[1].nAnalogInput <-> TxPDO 5/Inputs/ADC-Value-ITV1
//     PlcTask Inputs/GVL_Hardware.aFbPneuChannel[2].nAnalogInput <-> TxPDO 5/Inputs/ADC-Value-ITV2
//     PlcTask Inputs/GVL_Hardware.aFbPneuChannel[3].nAnalogInput <-> TxPDO 5/Inputs/ADC-Value-ITV3
//     PlcTask Outputs/GVL_Hardware.aFbPneuChannel[1].nAnalogOutput <-> RxPDO 5/Outputs/DAC-Value-ITV1
//     PlcTask Outputs/GVL_Hardware.aFbPneuChannel[2].nAnalogOutput <-> RxPDO 5/Outputs/DAC-Value-ITV2
//     PlcTask Outputs/GVL_Hardware.aFbPneuChannel[3].nAnalogOutput <-> RxPDO 5/Outputs/DAC-Value-ITV3
//     PlcTask Outputs/GVL_Hardware.aPumps[2].bDigiOut <-> RxPDO 1/Outputs/Output-Ctrl_2
//     PlcTask Outputs/GVL_Hardware.aPumps[2].bDigiOut <-> RxPDO 1/Outputs/Output-Ctrl_7
//     PlcTask Outputs/GVL_Hardware.aPumps[3].bDigiOut <-> RxPDO 1/Outputs/Output-Ctrl_8
//     PlcTask Outputs/GVL_Hardware.aPumps[2].nPWMValue <-> RxPDO 10/Outputs/Output-Pulse_7
//     PlcTask Outputs/GVL_Hardware.fbPCV.bDigiOut <-> RxPDO 1/Outputs/Output-Ctrl_1
//     PlcTask Outputs/GVL_Hardware.fbPCV.bDigiOut <-> RxPDO 1/Outputs/Output-Ctrl_6
//     PlcTask Outputs/GVL_Hardware.fbPCV.bPneuValve <-> RxPDO 1/Outputs/Output-Ctrl_3
//   SPS1/SPS1 Instance <-> Device 3 (EtherCAT)/-KL01 (EK1100)/-KL07 (EL1918)
//     PlcTask Inputs/GVL_Hardware.fbSafety.bBoxContactsClosed <-> Device Info Data/Internal I/O/Input Safe Data FSIN Module 6.Input
//     PlcTask Inputs/GVL_Hardware.fbSafety.bDriveIsSafe <-> StandardInputs/Standard Out Var 25
//     PlcTask Inputs/GVL_Hardware.fbSafety.bEmergencyStop <-> StandardInputs/Standard Out Var 13
//     PlcTask Inputs/GVL_Hardware.fbSafety.bInterlockIsLocked <-> Device Info Data/Internal I/O/Input Safe Data FSIN Module 5.Input
//     PlcTask Inputs/GVL_Hardware.fbSafety.bMesIsSafe <-> StandardInputs/Standard Out Var 24
//     PlcTask Inputs/GVL_Hardware.fbSafety.nTwinSafeGrpState <-> TwinSAFE Group Info Data/TwinSafeGroup1 Info Data/State
//     PlcTask Outputs/GVL_Hardware.fbSafety.bErrAckTwinSafeGrp <-> StandardOutputs/Standard In Var 1
//     PlcTask Outputs/GVL_Hardware.fbSafety.bRequDriveOn <-> StandardOutputs/Standard In Var 11
//     PlcTask Outputs/GVL_Hardware.fbSafety.bRequMesOn <-> StandardOutputs/Standard In Var 12
//     PlcTask Outputs/GVL_Hardware.fbSafety.bRequUnlock <-> StandardOutputs/Standard In Var 14
//     PlcTask Outputs/GVL_Hardware.fbSafety.bRunStopTwinSafeGrp <-> StandardOutputs/Standard In Var 23
//   SPS1/SPS1 Instance <-> Device 3 (EtherCAT)/Drive1 (C1250-DS-XC-1S)X
//     PlcTask Inputs/GVL_Hardware.fbX1DriveLmtDS.nCapturedCounter <-> User Defined Inputs/Captured Counter
//     PlcTask Inputs/GVL_Hardware.fbX1DriveLmtDS.nCapturedValue <-> User Defined Inputs/Captured Value
//     PlcTask Inputs/GVL_Hardware.fbX1DriveLmtDS.nErrorCode <-> User Defined Inputs/ErrorCode
//     PlcTask Inputs/GVL_Hardware.fbX1DriveLmtDS.nStatusWord <-> User Defined Inputs/Status Word
//     PlcTask Inputs/GVL_Hardware.stTipCalibrator.bXSensor <-> User Defined Inputs/X4 Inputs
//   SPS1/SPS1 Instance <-> Device 3 (EtherCAT)/Drive2 (C1250-DS-XC-1S)Y
//     PlcTask Inputs/GVL_Hardware.fbY1DriveLmtDS.nCapturedCounter <-> User Defined Inputs/Captured Counter
//     PlcTask Inputs/GVL_Hardware.fbY1DriveLmtDS.nCapturedValue <-> User Defined Inputs/Captured Value
//     PlcTask Inputs/GVL_Hardware.fbY1DriveLmtDS.nErrorCode <-> User Defined Inputs/ErrorCode
//     PlcTask Inputs/GVL_Hardware.fbY1DriveLmtDS.nStatusWord <-> User Defined Inputs/Status Word
//     PlcTask Inputs/GVL_Hardware.stTipCalibrator.bYSensor <-> User Defined Inputs/X4 Inputs
//   SPS1/SPS1 Instance <-> NC-Task 1 SAF/Axes/Achse 1 (X)
//     PlcTask Inputs/GVL_Hardware.AxisRefX1.NcToPlc <-> Outputs/ToPlc
//     PlcTask Outputs/GVL_Hardware.AxisRefX1.PlcToNc <-> Inputs/FromPlc
//   SPS1/SPS1 Instance <-> NC-Task 1 SAF/Axes/Achse 2 (Y)
//     PlcTask Inputs/GVL_Hardware.AxisRefY1.NcToPlc <-> Outputs/ToPlc
//     PlcTask Outputs/GVL_Hardware.AxisRefY1.PlcToNc <-> Inputs/FromPlc
//   SPS1/SPS1 Instance <-> NC-Task 1 SAF/Axes/Achse 4 Q1
//     PlcTask Inputs/GVL_Hardware.AxisRefQ1.NcToPlc <-> Outputs/ToPlc
//     PlcTask Outputs/GVL_Hardware.AxisRefQ1.PlcToNc <-> Inputs/FromPlc
//   SPS1/SPS1 Instance <-> NC-Task 1 SAF/NC Kanal
//     GCodeTask Inputs/GCode.stGCodeRef.sNciToPlc <-> Outputs/ToPlc
//     GCodeTask Outputs/GCode.stGCodeRef.sPlcToNci <-> Inputs/FromPlc

CONFIGURATION SPS1
    RESOURCE PLC ON TwinCAT3
        TASK ComTask(INTERVAL := T#4ms, PRIORITY := 8);
        TASK GCodeTask(INTERVAL := T#2ms, PRIORITY := 6);
        TASK PlcTask(INTERVAL := T#10ms, PRIORITY := 14);
        PROGRAM CANInterfaceCom WITH ComTask : CANInterfaceCom;
        PROGRAM SerialBackCom WITH ComTask : SerialBackCom;
        PROGRAM FirmwUpdate WITH ComTask : FirmwUpdate;
        PROGRAM GCode WITH GCodeTask : GCode;
        PROGRAM MAIN WITH PlcTask : MAIN;
    END_RESOURCE
END_CONFIGURATION

// ---- Configuration/ST_IdNode.TcDUT
TYPE ST_IdNode :
STRUCT
	nId : UINT;
	pNext : POINTER TO ST_IdNode;
END_STRUCT
END_TYPE

// ---- DUTs/Enums/E_ActionStatus.TcDUT
TYPE E_ActionStatus :
(
	ACTIONSTATUS_Idle := 0,
	ACTIONSTATUS_Active,
	ACTIONSTATUS_PauseRequest,
	ACTIONSTATUS_Pause,
	ACTIONSTATUS_Ready,
	ACTIONSTATUS_Error
)USINT;
END_TYPE

// ---- DUTs/Enums/E_ArrayOrder.TcDUT
TYPE E_ArrayOrder :
(
	RowWiseSaw,
	RowWiseMeander,
	ColWiseSaw,
	ColWiseMeander
)USINT;
END_TYPE

// ---- DUTs/Enums/E_Condition.TcDUT
TYPE E_Condition :
(
	CONDITION_Nothing := 0,
	CONDITION_PreStepReady,
	CONDITION_SpecStepReady,
	CONDITION_ProcessVarGEQ,
	CONDITION_ProcessVarLEQ,
	CONDITION_UserInput,
	CONDITION_StepResult
)USINT;
END_TYPE

// ---- DUTs/Enums/E_CrashAvoidanceMode.TcDUT
{attribute 'qualified_only'}
TYPE E_CrashAvoidanceMode :
(
	MoveAllFree := 0,	//Es werden alle Tools bis zur FreeHeight freigefahren
	MoveNoneFree := 1,	//Es erfolgt keine Überprüfung (sollte nur intern in ComplexActions genutzt werden)
	MoveUnusedFree := 2	//Es werden alle anderen Tools freigefahren, beim benutzten Tool werden die Targets im Verfahrbereich gecheckt
)USINT;
END_TYPE

// ---- DUTs/Enums/E_DilPrepareMode.TcDUT
TYPE E_DilPrepareMode :
(
	ForAspirate := 0,
	ForDispense := 1
)USINT;
END_TYPE

// ---- DUTs/Enums/E_DilPumpMode.TcDUT
TYPE E_DilPumpMode :
(
	MODE_Suck := 0,
	MODE_Press := 1
)USINT;
END_TYPE

// ---- DUTs/Enums/E_DilType.TcDUT
TYPE E_DilType :
(
	DILTYPE_Single := 0,
	DILTYPE_TwinParallel := 1,
	DILTYPE_TwinSerial := 2,
	DILTYPE_TwinTransfer := 3
)USINT;
END_TYPE

// ---- DUTs/Enums/E_DilValveType.TcDUT
TYPE E_DilValveType :
(
	VALVETYPE_UNDEFINED := 0,
	VALVETYPE_3Way := 1,
	VALVETYPE_4Distribution := 10
)USINT;
END_TYPE

// ---- DUTs/Enums/E_DispenserState.TcDUT
TYPE E_DispenserState :
(
	Idle,
	Preparing,
	Dispensing
)USINT;
END_TYPE

// ---- DUTs/Enums/E_DrivingPinCtrl.TcDUT
{attribute 'qualified_only'}
TYPE E_DrivingPinCtrl :
(
	Horizontal,
	Vertical
)USINT;
END_TYPE

// ---- DUTs/Enums/E_DrivingPinSelection.TcDUT
{attribute 'qualified_only'}
TYPE E_DrivingPinSelection :
(
	Both,
    Left,
    Right
)USINT;
END_TYPE

// ---- DUTs/Enums/E_DrivingPinState.TcDUT
{attribute 'qualified_only'}
TYPE E_DrivingPinState :
(
	UNDEFINED := 0,
	Horizontal,
	Vertical
)USINT;
END_TYPE

// ---- DUTs/Enums/E_ErrorIdDS402.TcDUT
TYPE E_ErrorIdDS402 :
(
	ERRORID_NoError							:= 0,
	ERRORID_NotReadyToSwitchOn				:= 42600,
	ERRORID_OperationNotEnabled				:= 42601,
	ERRORID_HomingInterruptedOrNotReached	:= 42602,
	ERRORID_FaultState						:= 42603
)UINT;
END_TYPE

// ---- DUTs/Enums/E_ErrorIdGCode.TcDUT
TYPE E_ErrorIdGCode :
(
	ERRORID_NoError					:= 0,
	ERRORID_InvalidToolNr			:= 42240,	//ToolNr muss zwischen 1 und 20 liegen
	ERRORID_InvalidRefObj			:= 42241,	//ungültiges Referenzobjekt
	ERRORID_NoSelectedTool			:= 42242, //im GCode kein Tool ausgewählt
	ERRORID_ZMoveOutsidePrintArea	:= 42243,  //es wurde versucht mit G00 Q1 bzw G01 Q1 außerhalb des Druckbereichs zu verfahren
	ERRORID_NciModuleNotAvailable	:= 42244,
	ERRORID_InvalidNciState			:= 42245,
	ERRORID_InvalidSequenceNr		:= 42246,	//muss derzeit zwischen 1-5 liegen
	ERRORID_ScaffoldHeightExceeded	:= 42247,
	ERRORID_InvalidPausePoint		:= 42248,
	ERRORID_ScaffoldWidthExceeded	:= 42249,
	ERRORID_ScaffoldDepthExceeded	:= 42250,
	ERRORID_InvalidRParameter		:= 42251,
	ERRORID_ToolIsNoUniDispenser	:= 42252
)UINT;
END_TYPE

// ---- DUTs/Enums/E_ErrorIdCan.TcDUT
TYPE E_ErrorIdCan :
(
	ERRORID_NoError					:= 0,
	ERRORID_NodeDeactivated			:= 42496,
	ERRORID_NodeNotFound			:= 42497,
	ERRORID_SdoSyntaxErrorAtStartup	:= 42498,
	ERRORID_SdoDataMismatchAtStartup:= 42499,
	ERRORID_NodePreOP				:= 42500,
	
	ERRORID_FileAlreadyOpened		:= 42512,
	ERRORID_FirmwFileCorrupt		:= 42513,
	ERRORID_FirmwFileCRCError		:= 42514,
	ERRORID_FirmwFileLineError		:= 42515,
	ERRORID_FirmwFileEOF			:= 42516,
	ERRORID_TimeoutSendCanMsg		:= 42517,
	
	ERRORID_XcpErrCmdSynch			:= 42528,
	ERRORID_XcpErrCmdBusy			:= 42529,
	ERRORID_XcpErrCmdUnknown		:= 42530,
	ERRORID_XcpErrOutOfRange		:= 42531,
	ERRORID_XcpErrAccessLocked		:= 42532,
	ERRORID_XcpErrPageNotValid		:= 42533,
	ERRORID_XcpErrSequence			:= 42534,
	ERRORID_XcpErrGeneric			:= 42535
	
)UINT;
END_TYPE

// ---- DUTs/Enums/E_ErrorIdHwGeneral.TcDUT
TYPE E_ErrorIdHwGeneral :
(
	ERRORID_NoError						:= 0,
	ERRORID_DriveNotHomed				:= 42100,
	ERRORID_InvalidPosition				:= 42101,
	ERRORID_InvalidSpeed				:= 42102,
	ERRORID_Timeout						:= 42103,
	ERRORID_InvalidHwRef				:= 42104,
	ERRORID_HomingFailed				:= 42105,
	ERRORID_PosOutsideToleranceWindow	:= 42106,
	ERRORID_TargetPosNotReached			:= 42107,
	ERRORID_UndefinedDriveError			:= 42108,
	ERRORID_HardwareNotEnabled			:= 42109,
	ERRORID_GenericError				:= 42110,
	ERRORID_MotorCurrentExceeded		:= 42111,
	ERRORID_InvalidInputVoltage			:= 42112,
	ERRORID_ControllerTemperature		:= 42113,
	ERRORID_InterlockError				:= 42114,
	ERRORID_SoftwareReset				:= 42115,
	ERRORID_InternalSoftwareError		:= 42116,
	ERRORID_InvalidRatedCurrent			:= 42117,
	ERRORID_BallastResistorOverloaded	:= 42118,
	ERRORID_MotorBlocked				:= 42119,
	ERRORID_InternalError				:= 42120,
	ERRORID_Sensor1Fault				:= 42121,
	ERRORID_Sensor2Fault				:= 42122,
	ERRORID_SensorNFault				:= 42123,
	ERRORID_MemoryError					:= 42124,
	ERRORID_FieldbusMonitoring			:= 42125,
	ERRORID_CANopenError				:= 42126,
	ERRORID_SpeedMonitoring				:= 42127,
	ERRORID_FollowingError				:= 42128,
	ERRORID_LimitSwitchExceeded			:= 42129,
	ERRORID_DriveIsInErrorState			:= 42130,
	ERRORID_DriveIsStillBusy			:= 42131,
	ERRORID_LockingFailed				:= 42132,
	ERRORID_UnlockingFailed				:= 42133
	
	
)UINT;
END_TYPE

// ---- DUTs/Enums/E_ExchangePieceOption.TcDUT
TYPE E_ExchangePieceOption :
(
	Slot := 0,
	NextSlotRespPiece := 1
)USINT;
END_TYPE

// ---- DUTs/Enums/E_ExtruderType.TcDUT
TYPE E_ExtruderType :
(
	PistonExtruder1,
	FilamentExtruder1,
	ScrewExtruder1,
	SyringeExtruder1,
	FilamentExtruder2,
	PureDyne_1,
	PureDyne_2,
	PureDyne_3
)USINT;
END_TYPE

// ---- DUTs/Enums/E_GCodeState.TcDUT
TYPE E_GCodeState :
(
	GCodeState_Idle := 0,
	GCodeState_Loading := 1,
	GCodeState_Starting := 2,
	GCodeState_Running := 3,
	GCodeState_PauseRequest := 4,
	GCodeState_Pause := 5,
	GCodeState_ContinueRequest := 6,
	GCodeState_Error := 99
)USINT;
END_TYPE

// ---- DUTs/Enums/E_GripperState.TcDUT
{attribute 'qualified_only'}
{attribute 'strict'}
TYPE E_GripperState :
(
	Undefined,
	Open,
	HalfClosed,
	FullyClosed
)USINT;
END_TYPE

// ---- DUTs/Enums/E_HardwarePropType.TcDUT
TYPE E_HardwarePropType :
(
	None := 0,
	RefPos1 := 1,
	RefPos2 := 2,
	HomePos := 3,
	AxisLength := 4,
	SliderLength := 5,
	InvertInitDir := 6,
	MinPos := 7,
	MaxPos := 8,
	LimitMargeNeg := 9,
	LimitMargePos := 10,
	MinSpeed := 11,
	MaxSpeed := 12,
	MinPress := 13,
	MaxPress := 14,
	MinPressCV := 15,
	MaxPressCV := 16,
	MinPressMV := 17,
	MaxPressMV := 18,
	FactorSetPress := 19,
	FactorCurrentPress := 20,
	WorkplateDim := 21,
	NullPosDist := 22,
	MaxPosDist := 23,
	SetupPosDist := 24,
	Disabled := 25,
	MinVoltage := 26,
	MaxVoltage := 27,
	MinVoltageCV := 28,
	MaxVoltageCV := 29,
	MinVoltageMV := 30,
	MaxVoltageMV := 31,
	MinCurrent := 32,
	MaxCurrent := 33,
	MinCurrentCV := 34,
	MaxCurrentCV := 35,
	FactorCurrentCV := 36,
	MinCurrentMV := 37,
	MaxCurrentMV := 38,
	FactorCurrentMV := 39,
	Legacy := 40,
	OffsetSetPress := 41,
	OffseCurrentPress := 42,
	DistPerMotorRev := 43,
	SlowHomingSpeed := 44,
	FastHomingSpeed := 45,
	HoldCurrent := 46
)UINT;
END_TYPE

// ---- DUTs/Enums/E_InteractMessageType.TcDUT
TYPE E_InteractMessageType :
(
	INTERACTMES_NONE := 0,
	INTERACTMES_StartObjRecog := 1,
	INTERACTMES_ObjRecogResult := 2,
	INTERACTMES_StartTeaching := 3,
	INTERACTMES_TeachingFinished := 4,
	INTERACTMES_MountZSensor := 5,
	INTERACTMES_UnmountZSensor := 6,
	INTERACTMES_Pause := 7,
	INTERACTMES_Continue := 8,
	INTERACTMES_Assume := 9,
	INTERACTMES_WaitForUser := 10,
	INTERACTMES_Cancel := 999
)UINT;
END_TYPE

// ---- DUTs/Enums/E_InterlockState.TcDUT
TYPE E_InterlockState :
(
	UNDEFINED,
	Unlocked,
	Locked,
	Error
)USINT;
END_TYPE

// ---- DUTs/Enums/E_CompOperator.TcDUT
{attribute 'qualified_only'}
TYPE E_CompOperator :
(
	COMP_OP_GT,	//>
	COMP_OP_LT,	//<
	COMP_OP_GE,	//>=
	COMP_OP_LE,	//<=
	COMP_OP_EQ,	//=
	COMP_OP_NE	//<>
)USINT;
END_TYPE

// ---- DUTs/Enums/E_LockCtrl.TcDUT
{attribute 'qualified_only'}
TYPE E_LockCtrl :
(
	Unlock,
	Lock
)USINT;
END_TYPE

// ---- DUTs/Enums/E_LockState.TcDUT
TYPE E_LockState :
(
	UNDEFINIED,
	Unlocked,
	Locked
)USINT;
END_TYPE

// ---- DUTs/Enums/E_MeasureMode.TcDUT
TYPE E_MeasureMode :
(
	MEAS_MODE_Auto := 0,
	MEAS_MODE_SemiAuto := 1
)USINT;
END_TYPE

// ---- DUTs/Enums/E_MeasureOption.TcDUT
TYPE E_MeasureOption :
(
	MEAS_OPTION_SlowApproach := 0,
	MEAS_OPTION_FastApproach := 1,
	MEAS_OPTION_OnlyXY := 2
)USINT;
END_TYPE

// ---- DUTs/Enums/E_MethodState.TcDUT
TYPE E_MethodState :
(
	Ready := 0,
	Busy := 1,
	Error := 2 
)USINT;
END_TYPE

// ---- DUTs/Enums/E_ModalDesignationAbsInc.TcDUT
TYPE E_ModalDesignationAbsInc :
(
	ModalDesignAbsInc_Undefined := 0,
	ModalDesignAbsInc_G90 := 4186,	//absolute designation
	ModalDesignAbsInc_G91 := 4187	//incremental designation
)UDINT;
END_TYPE

// ---- DUTs/Enums/E_ModalGeoTypes.TcDUT
TYPE E_ModalGeoTypes :
(
	MODALGEOTYPE_Undefined := 0,
	MODALGEOTYPE_G0 := 4096,
	MODALGEOTYPE_G01 := 4097,
	MODALGEOTYPE_G02 := 4098,
	MODALGEOTYPE_G03 := 4099
)UDINT;
END_TYPE

// ---- DUTs/Enums/E_MoveDirection.TcDUT
TYPE E_MoveDirection :
(
	DIRECTION_STOP := 0,
	DIRECTION_XPLUS := 1,
	DIRECTION_XMINUS := 2,
	DIRECTION_YPLUS := 3,
	DIRECTION_YMINUS := 4,
	DIRECTION_ZPLUS := 5,
	DIRECTION_ZMINUS := 6
)USINT;
END_TYPE

// ---- DUTs/Enums/E_MoveMode.TcDUT
TYPE E_MoveMode :
(
	MODE_Relative 				:= 0,
	MODE_AbsWithOffset			:= 1,
	MODE_AbsNoneOffset 			:= 2,
	MODE_Free					:= 3,	//nur für Z-Ache
	MODE_Home					:= 4,	//nur für Z-Ache
	MODE_Measure				:= 5	//nur für Z-Achse mit ZLevelSensor
)USINT;
END_TYPE

// ---- DUTs/Enums/E_ObjectGroup.TcDUT
TYPE E_ObjectGroup :
(
	OBJECTGROUP_Undefined := 0,
	OBJECTGROUP_Device := 1,
	OBJECTGROUP_Target := 2,
	OBJECTGROUP_MzTool := 4,
	OBJECTGROUP_Piece := 8,
	OBJECTGROUP_Rack := 16,
	OBJECTGROUP_Array := 32,
	OBJECTGROUP_GCodeTool := 64
)USINT;
END_TYPE

// ---- DUTs/Enums/E_OpClCtrl.TcDUT
TYPE E_OpClCtrl :
(
	Open,
	Close
)USINT;
END_TYPE

// ---- DUTs/Enums/E_OpClState.TcDUT
TYPE E_OpClState :
(
	UNDEFINED,
	Closed,
	Open
)USINT;
END_TYPE

// ---- DUTs/Enums/E_LogicOperator.TcDUT
{attribute 'qualified_only'}
TYPE E_LogicOperator :
(
	LOGIC_OP_UNDEFINED := 0,
	LOGIC_OP_AND := 1,
	LOGIC_OP_OR := 2
)USINT;
END_TYPE

// ---- DUTs/Enums/E_PickPutMode.TcDUT
TYPE E_PickPutMode :
(
	MODE_Pick := 0,
	MODE_Put := 1
)USINT;
END_TYPE

// ---- DUTs/Enums/E_POU.TcDUT
TYPE E_POU :
(
	POU_UNDEFIEND := 0,
	POU_FB_DeviceBase,
	POU_FB_Diluter,
	POU_FB_InkStation,
	POU_FB_LiquidReserve,
	POU_FB_MtpHolder,
	POU_FB_PowderStation,
	POU_FB_Reactor,
	POU_FB_Stroboscope,
	POU_FB_SubstHolder,
	POU_FB_TipCalibrator,
	POU_FB_TipCleaner,
	POU_FB_WashStation,
	POU_FB_Camera,
	POU_FB_CartDispenser,
	POU_FB_MultiCartHolder,
	POU_FB_DeloDot,
	POU_FB_Exposure,
	POU_FB_FlipTubeHandler,
	POU_FB_Luer,
	POU_FB_MzBase,
	POU_FB_MzHead,
	POU_FB_MzTool,
	POU_FB_PassivPip,
	POU_FB_PiezoPip,
	POU_FB_Pipette,
	POU_FB_PowderPip,
	POU_FB_StampSupport,
	POU_FB_TriplePip,
	POU_FB_ZLevelSensor,
	POU_FB_FlipTube,
	POU_FB_NeedleTip,
	POU_FB_Piece,
	POU_FB_Septum,
	POU_FB_Stamp,
	POU_FB_UsingPiece,
	POU_FB_Vial,
	POU_FB_DryPad,
	POU_FB_FlipTubeRack,
	POU_FB_Mtp,
	POU_FB_NeedleRack,
	POU_FB_PortRack,
	POU_FB_Rack,
	POU_FB_SeptumRack,
	POU_FB_SeptumWaste,
	POU_FB_Slide,
	POU_FB_SpotPattern,
	POU_FB_StampMagazine,
	POU_FB_TargetBase,
	POU_FB_TargetTray,
	POU_FB_TipRack,
	POU_FB_VialRack,
	POU_FB_Wafer,
	POU_FB_ObjectManagment,
	POU_PC_Control,
	POU_MAIN,
	POU_FB_ActionDispacher,
	POU_FB_ComplexAction,
	POU_GCode,
	POU_FB_GCodeSwitchPress,
	POU_FB_MeasTip,
	POU_FB_SM_Auto,
	POU_FB_SM_Config,
	POU_FB_SM_Init,
	POU_FB_SM_Maintenance,
	POU_FB_SM_Manu,
	POU_FB_SM_Mode,
	POU_FB_SM_SemiAuto,
	POU_FB_MultiZRef,
	POU_FB_HwRef4ChHeater,
	POU_FB_HwRefBottleRack,
	POU_FB_HwRefIOExpander,
	POU_FB_HwRefReactHeater,
	POU_FB_HwRefTripleTrigger,
	POU_FB_HskMFunc,
	POU_FB_Sequenece,
	POU_FB_TwinPiezoHolder,
	POU_FB_Configuration,
	POU_FB_Extruder,
	POU_ScanHwModules,
	POU_PrepareHwModules,
	POU_FB_pHElectrode,
	POU_FB_pHElectrodeCap,
	POU_FB_pHElectrodeCapRack,
	POU_FB_TitrationTool,
	POU_FB_TwinExtruder,
	POU_FB_Safety,
	POU_FB_HighVoltTray,
	POU_FB_VacuumHandler,
	POU_FB_VermesDisp,
	POU_FB_CustomUnitType1,
	POU_FB_HybridDispenser,
	POU_FB_CustomUnitType2,
	POU_FB_Gripper,
	POU_FB_TrayTransporter,
	POU_FB_Stacker,
	POU_FB_HwRefNanotecPD
)UINT;
END_TYPE

// ---- DUTs/Enums/E_POUACT.TcDUT
TYPE E_POUACT :
(
	POUACT_UNDEFIEND := 0,
	POUACT_A_Init,
	POUACT_A_MovePlunger,
	POUACT_A_MoveValve,
	POUACT_A_Pump,
	POUACT_A_Reset,
	POUACT_A_Stop,
	POUACT_A_OpenClose,
	POUACT_A_Spin,
	POUACT_A_EmptyLiquid,
	POUACT_A_EmptyWaste,
	POUACT_A_FillLiquid,
	POUACT_A_Leveling,
	POUACT_A_Reload,
	POUACT_A_Shaking,
	POUACT_A_Cooling,
	POUACT_A_DetectVial,
	POUACT_A_StrobTest,
	POUACT_A_Heating,
	POUACT_A_SetPress,
	POUACT_A_SwitchPress,
	POUACT_A_SetPressCore,
	POUACT_A_SetPressShell,
	POUACT_A_SwitchPressCore,
	POUACT_A_SwitchPressShell,
	POUACT_A_Dispense,
	POUACT_A_InitSpec,
	POUACT_A_Expose,
	POUACT_A_Aspirate,
	POUACT_A_Eject,
	POUACT_A_JogXY,
	POUACT_A_MoveX,
	POUACT_A_MoveXY,
	POUACT_A_MoveY,
	POUACT_A_MoveZ,
	POUACT_A_MoveChildsFree,
	POUACT_A_JogZ,
	POUACT_A_DispensePiezo,
	POUACT_A_PickPut,
	POUACT_A_PulsePress,
	POUACT_A_Adjust,
	POUACT_A_LockUnlock,
	POUACT_A_Cancel,
	POUACT_A_CalibrateZSensor,
	POUACT_A_CleanTip,
	POUACT_A_DockTool,
	POUACT_A_DryPip,
	POUACT_A_ExchangeNeedle,
	POUACT_A_ExchangeSeptum,
	POUACT_A_ExchangeStamp,
	POUACT_A_ExchangeTip,
	POUACT_A_ExchangeVial,
	POUACT_A_GetPipSample,
	POUACT_A_InsertTool,
	POUACT_A_MeasureStamp,
	POUACT_A_MeasureTarget,
	POUACT_A_MeasureTool,
	POUACT_A_MoveToTarget,
	POUACT_A_OpenCloseFlipTube,
	POUACT_A_RunGCode,
	POUACT_A_StampDemold,
	POUACT_A_StampInking,
	POUACT_A_TeachTarget,
	POUACT_A_TeachTool,
	POUACT_A_DispenseTest,
	POUACT_A_WashTool,
	POUACT_A_AssignRParamHeader,
	POUACT_A_BuildGroup,
	POUACT_A_Clean_MeasureTip,
	POUACT_A_ClearGroup,
	POUACT_A_Continue,
	POUACT_A_DispensePiezoInWaste,
	POUACT_A_HskMFunc,
	POUACT_A_MoveZHome,
	POUACT_A_Pause,
	POUACT_A_Run,
	POUACT_A_SelectTool,
	POUACT_A_WaitAtPoint,
	POUACT_A_WaitForUser,
	POUACT_A_WashDryPip,
	POUACT_A_MeasureX,
	POUACT_A_MeasureY,
	POUACT_A_MeasureZ,
	POUACT_A_ProbeX,
	POUACT_A_ProbeY,
	POUACT_A_Activate,
	POUACT_A_CheckObjProps,
	POUACT_A_CxGetDeviceIdent,
	POUACT_A_SetConfig,
	POUACT_A_SetConfigLegacy,
	POUACT_A_SetupAxis,
	POUACT_A_SetupDefaultObj,
	POUACT_A_SetupHardware,
	POUACT_A_DeviceFirmwUpdate,
	POUACT_A_SwitchPump,
	POUACT_A_Rinse,
	POUACT_A_DelConfig,
	POUACT_A_TransferGas,
	POUACT_A_TransferLiquid,
	POUACT_A_ActionOnArray,
	POUACT_A_Monitor,
	POUACT_A_Load,
	POUACT_A_Start,
	POUACT_A_Sequence,
	POUACT_A_Swivel,
	POUACT_A_MoveAllHome,
	POUACT_A_Extrude,
	POUACT_A_Prepare,
	POUACT_A_ExchangepHCap,
	POUACT_A_MeasurepH,
	POUACT_A_Mix,
	POUACT_A_Lock,
	POUACT_A_Unlock,
	POUACT_A_RunWithBoxContacts,
	POUACT_A_RunWithoutBoxContacts,
	POUACT_A_DilMoveValve,
	POUACT_A_SetPrintParams,
	POUACT_A_BasicDispense,
	POUACT_A_CleanTipGen2,
	POUACT_A_PipPreSequence,
	POUACT_A_PipPostSequence,
	POUACT_A_StirrCartridge,
	POUACT_A_UniDispense,
	POUACT_A_ExchangeVialGripper,
	POUACT_A_MoveSlider,
	POUACT_A_TurnDrivingPin,
	POUACT_A_TransferTray,
	POUACT_A_TransferTrayLeftToSlot,
	POUACT_A_TransferTrayRightToSlot,
	POUACT_A_TransferTraySlotToLeft,
	POUACT_A_TransferTraySlotToRight,
	POUACT_A_TurnTo,
	POUACT_A_OpClTrayStop,
	POUACT_A_MoveLifter
)UINT;
END_TYPE

// ---- DUTs/Enums/E_PressCtrl.TcDUT
TYPE E_PressCtrl :
(
	PRESSCTRL_Off := 0,
	PRESSCTRL_PressOn := 1,
	PRESSCTRL_VacOn := 2,
	PRESSCTRL_BothOn := 3,
	PRESSCTRL_UNDEFINED := 99
)USINT;
END_TYPE

// ---- DUTs/Enums/E_PrintParamType.TcDUT
TYPE E_PrintParamType :
(
	Undefined,
	Pressure,
	Feed,
	Flow,
	Frequency,
	Pulse,
	Voltage
)USINT;
END_TYPE

// ---- DUTs/Enums/E_ProcDataType.TcDUT
TYPE E_ProcDataType :
(
	PROCDATATYPE_Temp1 := 0,
	PROCDATATYPE_Temp2 := 1,
	PROCDATATYPE_Press1 := 2,
	PROCDATATYPE_Press2 := 3,
	PROCDATATYPE_Voltage1 := 4,
	PROCDATATYPE_Voltage2 := 5,
	PROCDATATYPE_Current1 := 6,
	PROCDATATYPE_Current2 := 7
)USINT;
END_TYPE

// ---- DUTs/Enums/E_StackerRotPosition.TcDUT
{attribute 'qualified_only'}
TYPE E_StackerRotPosition :
(
	UNDEFINED,
	LoadingPosition,
	TransferPositionPrinter1,
	TransferPositionPrinter2
)USINT;
END_TYPE

// ---- DUTs/Enums/E_SwivelCtrl.TcDUT
TYPE E_SwivelCtrl :
(
	Original,
    Swiveled
)USINT;
END_TYPE

// ---- DUTs/Enums/E_SwivelState.TcDUT
TYPE E_SwivelState :
(
	UNDEFINED,
    Original,
    Swiveled
)USINT;
END_TYPE

// ---- DUTs/Enums/E_TargetRef.TcDUT
TYPE E_TargetRef :
(
	TARGETREF_UNFEFINED := 0,
	TARGETREF_LeftBottom,
	TARGETREF_LeftTop,
	TARGETREF_RightTop,
	TARGETREF_RightBottom,
	TARGETREF_Center,
	TARGETREF_SpecPoint,
	TARGETREF_TwoDimArray,
	TARGETREF_NextPoint,
	TARGETREF_Slot,
	TARGETREF_Alignment,
	TARGETREF_SequParaToArrayItem
)USINT;
END_TYPE

// ---- DUTs/Enums/E_Action.TcDUT
TYPE E_Action :
(
	ACTION_Nothing 				:= 0,
	ACTION_RunGCode	 			:= 1,
	ACTION_ShiftGCodeZPos		:= 2,
	ACTION_Delay 				:= 6,
	ACTION_GoToStep				:= 7,
	ACTION_PauseStep			:= 8,
	ACTION_CounterStep			:= 9,
	ACTION_RunSequence			:= 10,
	ACTION_CoupleHeads			:= 11,	//untere Y-Achse mir der Oberen Y-Achse koppeln
	
	ACTION_Init 				:= 50,
	ACTION_DilMovePlunger 		:= 51,
	ACTION_DilMoveValve 		:= 52,
	ACTION_DilPump		 		:= 53,
	ACTION_DilTransfer	 		:= 54,
	ACTION_DilPrepare	 		:= 55,	//Reload und MoveValve für Aspirieren bzw Dispensen
	ACTION_SetVacuum			:= 56,
	ACTION_SuckOff				:= 57,
	ACTION_Jog 					:= 58,
	ACTION_MoveX 				:= 59,
	ACTION_MoveY 				:= 60,
	ACTION_MoveXY 				:= 61,
	ACTION_MoveZ 				:= 62,
	ACTION_Heating 				:= 63,
	ACTION_Cooling 				:= 64,
	ACTION_SwitchLight			:= 65,
	ACTION_InkSpin				:= 66,
	ACTION_InkOpClCover			:= 67,	//Deckel Inkstation auf/zu
	ACTION_PowdStatReload 		:= 68,	//Stößel der PowderStation nach unten fahren zum Nachfüllen
	ACTION_PowdStatShaking 		:= 69,	//Pulver schütteln
	ACTION_PowdStatLeveling 	:= 70,	//Pulver nivellieren
	ACTION_SetPressure			:= 71,	//Druck einstellen
	ACTION_SwitchPressure		:= 72,	//Druck/Vakuum schalten
	ACTION_PulsePressure		:= 73,	//zwei Druckkanäle alternierend schalten
	ACTION_SwitchPump			:= 74,	//Pumpen ein/aus (Waschstation(Waste,Rinse), PiezoPip->Druckausgleichsbehälter)
	ACTION_OpenClose			:= 75,	//Öffnen/Schließen
	ACTION_LockUnlock			:= 76,	//Tool verriegeln, entriegeln (Stampsupport, Extruder)
	ACTION_StampAdjust			:= 77,	//Stempel drehen
	ACTION_Aspirate				:= 78,	//mit einem MzTool aspirieren
	ACTION_Dispense				:= 79,	//mit einem MzTool dispensen
	ACTION_DispenseDrops		:= 80,	//mit einer PiezoPipette oder einem Delo dispensen
	ACTION_StrobTest			:= 81,	//das Stroboskop mit 125Hz triggern (zu Testzwecken)
	ACTION_ChangeCleanMat		:= 82,	//Reinigungsmaterial gewechselt (Drypad, TipCleaner)
	ACTION_EmptyWaste			:= 83,	//ein Device leeren (z.B. Waschsation)
	ACTION_Rinse				:= 84,	//Waschstation Spülung
	ACTION_Eject				:= 85,	//Eject
	ACTION_Expose				:= 86,	//Expose
	ACTION_PickPutPowder		:= 87,	//Pulver mit einer PulverPipette aufnehmen/abgeben
	ACTION_ReactorOpCl			:= 88,	//Reaktor -Klemme, Deckel öffnen/schließen
	ACTION_DetectVial			:= 89,	//Detektion des Reaktor-Vials veranlassen
	ACTION_FillLiquid			:= 90,	//ein Device befüllen
	ACTION_EmptyLiquid			:= 91,	//ein Device leeren
	ACTION_Swivel				:= 92,	//TwinPipHolder schwenken
	ACTION_SetVoltage			:= 93,	//Hochspannung einstellen
	ACTION_SwitchVoltage		:= 94,	//Hochspannung einschalten
	ACTION_Extrude				:= 95,	//Extrudieren
	ACTION_ExtrMovePlunger		:= 96,	//Kolben eines Pistonextruders zu bestimmter Position fahren
	ACTION_Mix					:= 97,	//abwechselnd Aspirieren/Dispensen mit einer Pipette oder Luer
	ACTION_MeasurepH			:= 98,	//MeasurepH
	ACTION_BasicDispense		:= 99,	//Dispenser Ein oder ausschalten ohne zusätliche Parameter
										//wir hauptsächlich vom Hybrid-Dispenser genutzt
									
	ACTION_StirrCartridge		:= 100,	//CartridgeStirrer EIN/AUS
	ACTION_TakePicture			:= 101,
	
	ACTION_TurnTo 				:= 103,
	ACTION_MoveLifter 			:= 104,
	ACTION_TurnDrivingPin		:= 105,
	ACTION_MoveTrayTransporter	:= 106,
	ACTION_LoadStacker			:= 107, 	//Be-und Entladen des Stackers
	
	ACTION_Stop 				:= 999,
	
	ACTION_MoveToTarget 		:= 1000,
	ACTION_MeasureTool			:= 1001,	//Vermessen (Tip oder ZLevel, ...)
	ACTION_OpenCloseFlipTube	:= 1002,
	
	ACTION_WashTool				:= 1007,	//Ein Tool an einer Waschststaion waschen
	ACTION_SetNcOverride		:= 1008,	//Unused
	ACTION_ExchangePiece		:= 1009,
	ACTION_StampDemolding		:= 1010,	//Stempel entformen
	ACTION_StampInking			:= 1011,	//mit Stempel Resist oder Ink-Substanz aufnehmen
	ACTION_CleanTip				:= 1012,	//Tip am TipCleaner reinigen
	//1013 ist obsolete - war mal WashSimple
	ACTION_DryPip				:= 1014,	//Pip an DryPad trocknen
	ACTION_DispenseTest			:= 1015,	//Piezo an an Stroboskop testen
	ACTION_TeachTarget			:= 1016,	//Ein Target mit einem MzTool einteachen
	ACTION_GetPipSample			:= 1017,	//Probe mit Pipette aufnehmen
	ACTION_CalibrateZSensor		:= 1018,	//ZSensor(MzTool) kalibrieren
	ACTION_TeachTool			:= 1019,	//MzTool anhand eines Referenztargets einteachen
	ACTION_InsertTool			:= 1020,	//MzTool in ein Target oder Piece (Vial, FlipTube) einführen bzw einstechen
	ACTION_DockTool				:= 1021,	//MzTool an ein Target oder Piece andocken
	ACTION_TransferLiquid		:= 1022,	//Liquid mittels Diluter von einem Luer zu einem zweiten Luer transferieren
	ACTION_TransferGas			:= 1023,	//Gas von einem Luer zu einem zweiten Luer transferieren
	ACTION_ActionOnArray		:= 1024,	//Ein spezielle Action nacheinander an jedem Index eines Arrays durchführen
	ACTION_DryToolInside		:= 1025,
	ACTION_MoveAllHome			:= 1026,
	ACTION_TransferTray			:= 1027		//Ein Tray mit einem TrayTransporter von oder zur Übergabestation transportieren
	
)UINT;
END_TYPE

// ---- DUTs/Enums/E_ErrorIdCmd.TcDUT
TYPE E_ErrorIdCmd :
(
	ERRORID_NoError := 0,
	//ERRORID_NoReply := 41472,
	ERRORID_WrongMode := 41473,
	ERRORID_ModeChangeImpossible := 41474,
	ERRORID_WrongObjecttype := 41475,
	ERRORID_ObjectNotExists := 41476,
	ERRORID_InvalidProperty := 41477,
	ERRORID_InvalidState := 41478,
	ERRORID_InvalidAction := 41479,
	//ERRORID_ObjectInUse := 41480,
	ERRORID_BasicActionActive := 41481,
	ERRORID_ComplexActionActive := 41482,
	ERRORID_InvalidHeatingTemp := 41483,
	ERRORID_InvalidTargetPointRef := 41484,
	ERRORID_InvalidTargetPointNr := 41485,
	ERRORID_InvalidTargetPointCol := 41486,
	ERRORID_InvalidTargetPointRow := 41487,
	ERRORID_PressTimeOut := 41488,
	ERRORID_InvalidPressure := 41489,
	ERRORID_InvalidMoveMode := 41490,
	ERRORID_DeviceNotInitialized := 41491,
	ERRORID_StepNotExists := 41492,
	ERRORID_StepHasNoBasicCondi := 41493,
	ERRORID_InvalidCondition := 41494,
	ERRORID_InvalidCondiOperator := 41495,
	ERRORID_PrestepNotExists := 41496,
	ERRORID_SpecstepNotExists := 41497,
	ERRORID_UnsuitableObject := 41498,
	ERRORID_UnsuitableTarget := 41499,
	ERRORID_TargetPosOutOfRangeX := 41500,
	ERRORID_VelocityOutOfRange := 41501,
	ERRORID_PipMoveWithZSensor := 41502,
	ERRORID_ConfigNotActivated := 41503,
	ERRORID_OnlyReadHwProp := 41504,
	ERRORID_UnknownMode := 41505,
	ERRORID_TipCalibSensor := 41506,
	ERRORID_TipCalibProbeSensorX := 41507,
	ERRORID_TipCalibProbeSensorY := 41508,
	ERRORID_InvalidWashMode := 41509,
	ERRORID_InvalidMeasureMode := 41510,
	ERRORID_ZSensorNotMounted := 41511,
	ERRORID_InkStationNotOpen := 41512,
	ERRORID_InkStationIsStillSpinning := 41513,
	ERRORID_VacuumNotOk := 41514,
	ERRORID_InkStatCoverAreaNotFree := 41515,
	ERRORID_InvalidPumpNr := 41516,
	ERRORID_InvalidDutyCycle := 41517,
	ERRORID_X2AxisNotCoupled := 41518,
	ERRORID_TimeOut := 41519,
	ERRORID_InvalidHwProperty := 41520,
	ERRORID_ToMuchFollwingSteps := 41521,
	ERRORID_InvalidSpecStep := 41522,
	ERRORID_InvalidDeviceForProcData := 41523,
	ERRORID_ToMuchActionsInActionDispacher := 41524,
	ERRORID_LiquidBottleEmpty := 41525,
	ERRORID_WasteBottleFull := 41526,
	ERRORID_TimeOutFillPCV := 41527,
	ERRORID_MissingSystemPressure := 41528,
	ERRORID_MeasureTouchProbeFail := 41529,
	ERRORID_MeasureZDistanceExeeded := 41530,
	ERRORID_InvalidHwGroup := 41531,
	ERRORID_InvalidHwItem := 41532,
	ERRORID_AxisStillBusy := 41533,
	ERRORID_SimultanErrorX1X2 := 41534,
	ERRORID_ZSensorNotCalibrated := 41535,
	ERRORID_NoPieceOnTool := 41536,
	ERRORID_PieceAlreadyOnTool := 41537,
	ERRORID_NoPieceInSlot := 41538,
	ERRORID_PieceAlreadyInSlot := 41539,
	ERRORID_InvalidStampAssignment := 41540,
	ERRORID_InvalidTargetSlot := 41541,
	ERRORID_SafetyBoxOpen := 41542,
	ERRORID_InvalidVoltageChannel := 41543,
	ERRORID_PieceAlreadyUsed := 41544,
	ERRORID_NoFreshPieceAvailable := 41545,
	ERRORID_NoFreeSlotAvailable := 41546,
	ERRORID_NoPieceDetermined := 41547,
	ERRORID_InvalidPieceType := 41548,
	ERRORID_InvalidCtrl := 41549,
	ERRORID_InvalidExchangeOption := 41550,
	ERRORID_FlipTubeAlreadyOpen := 41551,
	ERRORID_FlipTubeNotOpen := 41552,
	ERRORID_SeptumAlreadyOnVial := 41553,
	ERRORID_NoVialInReactor := 41554,
	ERRORID_VialAlreadyInReactor := 41555,
	ERRORID_AnyToolNotCrashSafe := 41556,
	ERRORID_ConfigErrorZSensor := 41557,
	ERRORID_InvalidLiquidChannel := 41558,
	ERRORID_InvalidWasteChannel := 41559,
	ERRORID_CoverNotClosed := 41560,
	ERRORID_CoverNotOpen := 41561,
	ERRORID_PowdDetectOnReloadPos := 41562,
	ERRORID_PowdLevelLow := 41563,
	ERRORID_ReactorNotOpen := 41564,
	ERRORID_ReactorCoverNotFree := 41565,
	ERRORID_NoNeedleOnTool := 41566,
	ERRORID_TargetPosOutOfRangeY := 41567,
	ERRORID_TargetPosOutOfRangeZ := 41568,
	ERRORID_JogDistanceRiskOfCrash := 41569,
	ERRORID_JogSpeedRiskOfCrash := 41570,
	ERRORID_PieceExchangeFailed := 41571,
	ERRORID_ErrorResetFailed := 41572,
	ERRORID_DeviceInErrorState := 41573,
	ERRORID_InvalidRinseChannel := 41574,
	ERRORID_StopButtonNotReleased := 41575,
	ERRORID_InterlockNotLocked := 41576,
	ERRORID_NotReadyToUnlock := 41577,
	ERRORID_SequenceNotExists := 41578,
	ERRORID_SequenceCannotCallItself := 41579,
	ERRORID_InvalidStepNr := 41580,
	ERRORID_StepAlreadyExists := 41581,
	ERRORID_StepNrExeedsMaxNoOfSteps := 41582,
	ERRORID_ActiveSequencesExeeded := 41583,
	ERRORID_ActionLocked := 41584,
	ERRORID_NoStepsInSequence := 41585,
	ERRORID_NoOfFollowerStepsExeeded := 41586,
	ERRORID_HighVoltSupplyOff := 41587,
	ERRORID_NotAllPipettesConfigured := 41588,
	ERRORID_MtpRowRiskOfCrash := 41589,
	ERRORID_NoFreeTimerAvailable := 41590,
	ERRORID_InvalidMeasureOption := 41591,
	ERRORID_MoveXYRiskOfCrash := 41592,
	ERRORID_InvalidCrashAvoidanceMode := 41593,
	ERRORID_InvalidFeed := 41594,
	ERRORID_DeviceAlreadyLocked := 41595,
	ERRORID_DeviceAlreadyUnLocked := 41596,
	ERRORID_DeviceNotLocked := 41597,
	ERRORID_RiskHighvoltFlashover := 41598,
	ERRORID_InvalidPlungerPos := 41599,
	ERRORID_CapOnElectrode := 41600,
	ERRORID_ToolHasNoEjector := 41601,
	ERRORID_WashStationHasNoAirShower := 41602,
	ERRORID_XAxisNotOnLeftLimitSwitch := 41603,
	ERRORID_InvalidTeachOption := 41604,
	ERRORID_InvalidSafetyState := 41605,
	ERRORID_TwinSafeGroupError := 41606,
	ERRORID_InterlockError := 41607,
	ERRORID_InvalidPrintParamType := 41608,
	ERRORID_InvalidArrayItem := 41609,
	ERRORID_OverCurrentHighVoltTray := 41610,
	ERRORID_NoCartridgeDispConfigured := 41611,
	ERRORID_NoExposureConfigured := 41612,
	ERRORID_PressureSupply := 41613,
	ERRORID_VacuumSupply := 41614,
	ERRORID_MoveZRiskOfCrash := 41615,
	ERRORID_InvalidSuckOffChannel := 41616,
	ERRORID_SensorAlreadySwitched := 41617,
	ERRORID_InvalidDiluterInput := 41618,
	ERRORID_InvalidActionDiluterType := 41619,
	ERRORID_NoTipCleanerConfigured := 41620,
	ERRORID_InvalidCleaningMode := 41621,
	ERRORID_InvalidCleaningWireSpeed := 41622,
	ERRORID_CalibrationPointHasAnOffset := 41623,
	ERRORID_InvalidPrintParamNumerator := 41624,
	ERRORID_TimeOutSuckOffLiquid := 41625,
	ERRORID_NotFullyOpened := 41626,
	ERRORID_NotFullyClosed := 41627,
	ERRORID_NoPieceTaken := 41628,
	ERRORID_ToolNotFreeOrBlocked := 41629,
	ERRORID_CouldNotOpenGripper := 41630,
	ERRORID_PieceNotInDestination := 41631,
	ERRORID_InvalidTarget := 41632,
	ERRORID_NotAvailable := 41633,
	ERRORID_DrivingPinLeftNotAvailable := 41634,
	ERRORID_DrivingPinRightNotAvailable := 41635,
	ERRORID_DrivingPinBlocked := 41636,
	ERRORID_NoTrayOnLeftTransferStation := 41637,
	ERRORID_NoTrayOnRightTransferStation := 41638,
	ERRORID_TrayAlreadyOnLeftTransferStation := 41639,
	ERRORID_TrayAlreadyOnRightTransferStation := 41640,
	ERRORID_CanNotTransferTrayCompletely := 41641,
	ERRORID_TransferAreaNotFree := 41642,
	ERRORID_TraysNotAligned := 41643,
	ERRORID_InvalidStackerAngle := 41644,
	ERRORID_TrayStopNotClosed := 41645,
	ERRORID_TrayStopNotOpen := 41646,
	ERRORID_StackerNotInTransferPosition := 41647,
	ERRORID_NoTrayInStackerShelf := 41648,
	ERRORID_TrayAlreadyInStackerShelf := 41649,
	ERRORID_StackerNotInShelfPosition := 41650
)UINT;
END_TYPE

// ---- DUTs/Enums/E_ErrorIdDiluter.TcDUT
TYPE E_ErrorIdDiluter :
(
	ERRORID_NoError					:= 0,
	ERRORID_ComTimeout				:= 41216,	//Kommunikationstimeout
	ERRORID_ReceiveDataError		:= 41217,	//Error beim Empfangen
	ERRORID_CecksumError			:= 41218,	//Error in der Antwort-Checksumme
	ERRORID_InitError				:= 41219,	//Error beim Initialisieren
	ERRORID_InvalidCommand			:= 41220,	//Fehlerhaftes Kommando übergeben
	ERRORID_InvalidOperand			:= 41221,	//Fehlerhafter Parameter übergeben
	ERRORID_InvalidCommandSeq		:= 41222,	//Fehlerhafte Kommandostruktur
	ERRORID_EepromFailure			:= 41223,	//Error im EEPROM
	ERRORID_NotIniialized			:= 41224, 	//Diluter nicht initialisiert
	ERRORID_PlungerOverload			:= 41225,	//Kolben ist blockiert
	ERRORID_ValveOverload			:= 41226,	//Ventil ist blockiert
	ERRORID_PlungerMoveNotAllowed	:= 41227,	//Kolben-Move nicht erlaubt
	ERRORID_CommandOverflow			:= 41228,	//Aktionskommando gesendet, bevor vorheriges abgearbeitet
	ERRORID_InvalidValveParam		:= 41229,	//Fehlerhafter Parameter für Ventilverstellung
	ERRORID_InvalidSyringe			:= 41230,	//Falsche Spritzgröße konfiguriert
	ERRORID_SpeedToSmall			:= 41231,	//Minimale Pumpgeschwindigkeit unterschritten
	ERRORID_SpeedExeeded			:= 41232,	//Maximale Pumpgeschwindigkeit überschritten
	ERRORID_InvalidPlungerPos		:= 41233,	//Kolbenposition ungültig
	ERRORID_InvalidValveType		:= 41234	//
)UINT;
END_TYPE

// ---- DUTs/Enums/E_ErrorIdMultiZ.TcDUT
TYPE E_ErrorIdMultiZ :
(
	ERRORID_NoError				:= 0,
	ERRORID_NoZAxis				:= 41728,	//ErrorCode MultiZ: "1"
	
	(*ERRORID_ReInitFail			:= 41729, //ErrorCode MultiZ: "2"
	ERRORID_LimitFail			:= 41730, //ErrorCode MultiZ: "3"
	ERRORID_InitLoop			:= 41731, //ErrorCode MultiZ: "4"
	ERRORID_StillMoving			:= 41732, //ErrorCode MultiZ: "5"
	ERRORID_ForceThresholdErr	:= 41733, //ErrorCode MultiZ: "6"
	ERRORID_PosAccuracy			:= 41734, //ErrorCode MultiZ: "7"
	ERRORID_InvalidTriggerVers	:= 41735, //ErrorCode MultiZ: "8"
	ERRORID_TipLimitFail		:= 41736, //ErrorCode MultiZ: "9"
	ERRORID_I2cTimeOutGen		:= 41737, //ErrorCode MultiZ: "10"
	ERRORID_TmcInvalidUdpateData:= 41738, //ErrorCode MultiZ: "11"
	ERRORID_TmcUdpateFailed		:= 41739, //ErrorCode MultiZ: "12"
	ERRORID_UnknownTool			:= 41740, //ErrorCode MultiZ: "13"
	ERRORID_I2cCommError		:= 41741, //ErrorCode MultiZ: "14"
	ERRORID_CommTimeoutMot		:= 41742, //ErrorCode MultiZ: "15"
	ERRORID_InvalidPiezoParam	:= 41743, //ErrorCode MultiZ: "16"
	ERRORID_AxisNotInitialized	:= 41744, //ErrorCode MultiZ: "17"
	ERRORID_NodePreop			:= 41745, //ErrorCode MultiZ: "18"
	ERRORID_ZSensSwitchFail		:= 41746, //ErrorCode MultiZ: "19"
	ERRORID_ZSensSwitchNotFound	:= 41747, //ErrorCode MultiZ: "20"
	ERRORID_No_Z_Limit			:= 41748, //ErrorCode MultiZ: "21"

	ERRORID_InvalidToolMode		:= 41750, //ErrorCode MultiZ: "23"
	
	ERRORID_GenericError		:= 41981, //ErrorCode MultiZ: "254"
	ERRORID_CommFailMot			:= 41982, //ErrorCode MultiZ: "255"*)
	
	ERRORID_ToResetErr				:= 41984,
	ERRORID_ToWaitSetPointAck		:= 41985,
	ERRORID_ToWaitTrgtReached		:= 41986,
	ERRORID_ToWaitStop				:= 41987,
	ERRORID_AxisNotHomed			:= 41988,
	ERRORID_TimeOutXYWaitInitZ		:= 41989,
	ERRORID_XYInitImpossible		:= 41990,
	ERRORID_InvalidZChannel			:= 41991,
	ERRORID_MultiZIsStillMoving		:= 41992,
	ERRORID_InvalidZAxisToolType	:= 41993,
	ERRORID_InvalidSdoVariType		:= 41994,
	ERRORID_InvalidToolConfig		:= 41995,
	ERRORID_InvalidHeaterConfig		:= 41996,
	ERRORID_TimeoutSwivel			:= 41997,
	ERRORID_TimeoutLock				:= 41998,
	ERRORID_TimeoutUnLock			:= 41999,
	ERRORID_TimeoutExtrude			:= 42000,
	ERRORID_TimeoutMovePlunger		:= 42001,
	ERRORID_FirmwareCartCoolerToLow := 42002,
	ERRORID_UnknownError			:= 65535
)UINT;
END_TYPE

// ---- DUTs/Enums/E_HardwareGrp.TcDUT
TYPE E_HardwareGrp :
(
	Nothing 				:= 0,
	AxisX					:= 1,
	AxisY					:= 2,
	MultiZBasis				:= 3,
	AxisZ					:= 4,
	Diluter					:= 5,
	PneuChannel				:= 6,
	Pump					:= 7,
	PCV						:= 8,
	MtpHeater				:= 9,
	SubstHeater				:= 10,
	ReactorHeater			:= 11,
	ReactorDrive			:= 12,
	BottleRack				:= 13,
	IOExpander				:= 14,
	TripleTrigger			:= 15,
	PowderStation			:= 16,
	InkStationSpinDrive		:= 17,
	InkStationCoverDrive	:= 18,
	TipCleaner				:= 19,
	Interlock				:= 20,
	StopButton				:= 21,
	EmergencyButton			:= 22,
	HighVoltSupply			:= 23,
	TMCM1140Stepper			:= 24,
	MultiPurpIO				:= 25,
	NanotecPD				:= 26,
	TMCM1140Stepper_Gen2	:= 27,
	EL70xx					:= 28
)UINT;
END_TYPE

// ---- DUTs/Enums/E_MachineMode.TcDUT
TYPE E_MachineMode :
(
	MACHINEMODE_UNDEFINED := 0,
	MACHINEMODE_Config,
	MACHINEMODE_Init,
	MACHINEMODE_Manu,
	MACHINEMODE_SemiAuto,
	MACHINEMODE_Auto,
	MACHINEMODE_Maintenance
)USINT;
END_TYPE

// ---- DUTs/Enums/E_MachineState.TcDUT
TYPE E_MachineState :
(
	MACHINESTATE_UNDEFINED := 0,
	MACHINESTATE_Idle,
	MACHINESTATE_Active,
	MACHINESTATE_PauseRequest,
	MACHINESTATE_Pause,
	MACHINESTATE_Cancel,
	MACHINESTATE_Canceled,
	MACHINESTATE_Ready,
	MACHINESTATE_Reset,
	MACHINESTATE_Running,
	MACHINESTATE_Error := 99
)USINT;
END_TYPE

// ---- DUTs/Enums/E_ObjectType.TcDUT
TYPE E_ObjectType :
(
	OBJECTTYPE_UNDEFINED 			:= 0,
	OBJECTTYPE_MZHead 				:= 1,
	OBJECTTYPE_PiezoPip 			:= 2,
	OBJECTTYPE_PassivPip 			:= 3,
	OBJECTTYPE_PowderPip 			:= 4,
	OBJECTTYPE_MultiCartHolder		:= 5,
	OBJECTTYPE_CartDispenser		:= 6,
	OBJECTTYPE_Camera 				:= 7,
	OBJECTTYPE_ZSensor 				:= 8,
	OBJECTTYPE_StampSupport			:= 9,
	OBJECTTYPE_Workplate 			:= 10,
	OBJECTTYPE_TipCleaner		 	:= 11,
	OBJECTTYPE_TipCalibrator	 	:= 12,
	OBJECTTYPE_WashStation 			:= 13,
	OBJECTTYPE_DryPad 				:= 14,
	OBJECTTYPE_Stroboscope 			:= 15,	
	OBJECTTYPE_MtpHolder 			:= 16,	
	OBJECTTYPE_SubstHolder 			:= 17,
	OBJECTTYPE_StampMagazine		:= 18,
	OBJECTTYPE_InkStation 			:= 19,
	OBJECTTYPE_PowderStation 		:= 20,
	OBJECTTYPE_TargetTray 			:= 21,
	OBJECTTYPE_Mtp 					:= 22,
	OBJECTTYPE_Slide 				:= 23,
	OBJECTTYPE_Wafer 				:= 24,
	OBJECTTYPE_Point 				:= 25,
	OBJECTTYPE_Diluter				:= 26,
	OBJECTTYPE_SpotArray			:= 27,
	OBJECTTYPE_DeloDot				:= 28,
	OBJECTTYPE_Exposure				:= 29,
	OBJECTTYPE_SpotPattern			:= 30,
	OBJECTTYPE_TargetGroup			:= 31,
	OBJECTTYPE_Stamp				:= 32,
	OBJECTTYPE_Needle				:= 33,
	OBJECTTYPE_Tip					:= 34,
	OBJECTTYPE_Vial					:= 35,
	OBJECTTYPE_VialClosed			:= 36,
	OBJECTTYPE_Septum				:= 37,
	OBJECTTYPE_Cartridge			:= 38,
	OBJECTTYPE_Port					:= 39,
	OBJECTTYPE_FlipTube				:= 40,
	OBJECTTYPE_TriplePip			:= 41,
	OBJECTTYPE_FlipTubeHandler		:= 42,
	OBJECTTYPE_Luer					:= 43,
	OBJECTTYPE_Reactor				:= 44,
	OBJECTTYPE_LiquidReserve		:= 45,
	OBJECTTYPE_SeptumWaste			:= 46,
	OBJECTTYPE_NeedleRack			:= 47,
	OBJECTTYPE_TipRack				:= 48,
	OBJECTTYPE_FlipTubeRack			:= 49,
	OBJECTTYPE_SeptumRack			:= 50,
	OBJECTTYPE_VialRack				:= 51,
	OBJECTTYPE_VialRackClosed		:= 52,
	OBJECTTYPE_PortRack				:= 53,
	OBJECTTYPE_VacuumHandler		:= 54,
	OBJECTTYPE_Nozzle				:= 55,
	OBJECTTYPE_SinglePiezoHolder	:= 56,
	OBJECTTYPE_TwinPiezoHolder		:= 57,
	OBJECTTYPE_HighVoltTray			:= 58,
	OBJECTTYPE_SolenoidPip			:= 59,
	OBJECTTYPE_Extruder				:= 60,
	OBJECTTYPE_pHElectrode			:= 61,
	OBJECTTYPE_pHElectrodeCap		:= 62,
	OBJECTTYPE_pHElectrodeCapRack	:= 63,
	OBJECTTYPE_TitrationTool		:= 64,
	OBJECTTYPE_WashTool				:= 65,
	OBJECTTYPE_TwinExtruder			:= 66,
	OBJECTTYPE_VermesDisp			:= 67,
	OBJECTTYPE_WorkplateCamera		:= 68,
	OBJECTTYPE_CartHolder			:= 69,
	OBJECTTYPE_DummyTool			:= 70,
	OBJECTTYPE_PassivePipGearPump	:= 71,
	OBJECTTYPE_CustomUnitType1		:= 72,
	OBJECTTYPE_HybridDispenser		:= 73,
	OBJECTTYPE_TipCleanerGen2		:= 74,
	OBJECTTYPE_CleaningBrush		:= 75,	
	OBJECTTYPE_Diluter3Inputs		:= 76,
	OBJECTTYPE_SubstHolderUnistat	:= 77,
	OBJECTTYPE_CartDispStirrer		:= 78,
	OBJECTTYPE_CustomUnitType2		:= 79,
	OBJECTTYPE_Gripper				:= 80,
	OBJECTTYPE_TrayTransporter		:= 81,
	OBJECTTYPE_PickPlacePip			:= 82,
	OBJECTTYPE_Stacker				:= 83
)UINT;
END_TYPE

// ---- DUTs/Enums/E_ErrorIdObjMgmt.TcDUT
TYPE E_ErrorIdObjMgmt :
(
	ERRORID_NoError 					:= 0,
	ERRORID_ObjectIdAlreadyExists 		:= 40960,	//Object mit dieser ID schon vorhanden
	ERRORID_InvalidObjectId 			:= 40961,	//Object mit dieser ID schon vorhanden
	ERRORID_CntObjectsExceeded 			:= 40962,	//Anzahl Objects überschritten
	ERRORID_CntDevicesExceeded 			:= 40963,	//Anzahl Devices überschritten
	ERRORID_CntTargetsExeeded 			:= 40964,	//Anzahl Targets überschritten
	ERRORID_CntMzToolsExceeded 			:= 40965,	//Anzahl MzTools überschritten
	ERRORID_CntMZHeadsExceeded 			:= 40966,	//Anzahl MzHeads überschritten
	ERRORID_CntPiezoPipsExceeded 		:= 40967,	//Anzahl PiezoPips überschritten
	ERRORID_CntPassivPipsExceeded 		:= 40968,	//Anzahl PassivPips überschritten
	ERRORID_CntPowderPipsExceeded 		:= 40969,	//Anzahl PowderPips überschritten
	ERRORID_CntCoreShellDispExceeded	:= 40970,	//Anzahl CoreShellDisp überschritten
	ERRORID_CntCartridgeDispExceeded	:= 40971,	//Anzahl CartridgeDisp überschritten
	ERRORID_CntCamerasExceeded			:= 40972,	//Anzahl Cameras überschritten
	ERRORID_CntZLevelSensorsExceeded	:= 40973,	//Anzahl ZLevelsensors überschritten
	ERRORID_CntStampSupportsExceeded	:= 40974,	//Anzahl StampSupports überschritten
	ERRORID_CntWorkplatesExceeded		:= 40975,	//Anzahl Workplates überschritten
	ERRORID_CntTipCleanerExceeded		:= 40976,	//Anzahl Tipcleaner überschritten
	ERRORID_CntTipCalibratorExceeded	:= 40977,	//Anzahl Tipcleaner überschritten
	ERRORID_CntWashStationsExceeded		:= 40978,	//Anzahl Washstations überschritten
	ERRORID_CntDrayPadsExceeded			:= 40979,	//Anzahl Drypads überschritten
	ERRORID_CntStroboscopesExceeded		:= 40980,	//Anzahl Stroboscopes überschritten
	ERRORID_CntMtpHoldersExceeded		:= 40981,	//Anzahl MtpHolder überschritten
	ERRORID_CntSubstHoldersExceeded		:= 40982,	//Anzahl SubstHolder überschritten
	ERRORID_CntStampHoldersExceeded		:= 40983,	//Anzahl SubstHolder überschritten
	ERRORID_CntInkStationsExceeded		:= 40984,	//Anzahl InkStations überschritten
	ERRORID_CntPowderStationsExceeded	:= 40985,	//Anzahl PowderStations überschritten
	ERRORID_CntSampleScannersExceeded	:= 40986,	//Anzahl SampleScanners überschritten
	ERRORID_CntTargetTraysExceeded		:= 40987,	//Anzahl TargetTrays überschritten
	ERRORID_CntMtpsExceeded				:= 40988,	//Anzahl Mtps überschritten
	ERRORID_CntSlidesExceeded			:= 40989,	//Anzahl Slides überschritten
	ERRORID_CntWafersExceeded			:= 40990,	//Anzahl Wafers überschritten
	ERRORID_CntPointsExceeded			:= 40991,	//Anzahl Points überschritten
	ERRORID_CntDilutersExceeded			:= 40992,	//Anzahl Diluters überschritten
	ERRORID_NotLastObject				:= 40993,	//Nicht das letzte Object
	ERRORID_InvalidObject				:= 40994,	//Object ungültig
	ERRORID_IsNoTarget					:= 40995,	//Object ist kein Target
	ERRORID_IsNoDevice					:= 40996,	//Object ist kein Device
	ERRORID_IsNoMzTool					:= 40997,	//Object ist kein MzTool
	ERRORID_InvalidParentTarget			:= 40998,	//ParentTarget ist kein gültiges Object
	ERRORID_ParentTargetIsNoTarget		:= 40999,	//ParentTarget ist kein Target
	ERRORID_InvalidParentMzTool			:= 41000,	//ParentMzTool ist kein gültiges Object
	ERRORID_ParentMzHeadIsNoMzHead		:= 41001,	//ParentMzHead ist kein MzHead 
	ERRORID_InvalidZAxisNr				:= 41002,	//ZAxisNr ungültig
	ERRORID_InvalidMultiZNr				:= 41003,	//MzHead akzeptiert nur 1 oder optional 2
	ERRORID_InvalidDiluterType			:= 41004,	//DiluterType ist ungültig
	ERRORID_InvalidDiluterChannel		:= 41005,	//DiluterChannel ist ungültig
	ERRORID_InvalidSyringeSize			:= 41006,	//Spritzgröße ist ungültig
	ERRORID_InvalidWorkplateNr			:= 41007,	//Workplate akzeptiert nur 1 oder optional 2
	ERRORID_InvalidPneuChannel			:= 41008,	//Pneumatikkanal nur zwischen 1 und 4 auswählbar
	ERRORID_InvalidMzDOutChannel		:= 41009,	//Digitaler Ausgang MzHead nur zwischen 1 und 8 auswählbar
	ERRORID_InvalidObjectType			:= 41010,	//Objecttyp ist ungültig
	ERRORID_InvalidHeaterChannel		:= 41011,	//ungültiger Heizerkanal
	ERRORID_InvalidDiluterObjId			:= 41012,	//angegebenes Objekt ist kein Diluter
	ERRORID_InvalidFrequency			:= 41013,	//Frequenz ungültig
	ERRORID_InvalidPulseWidth			:= 41014,	//Pulsbreite ungültig
	ERRORID_InvalidVoltage				:= 41015,	//Piezospannung ungültig
	ERRORID_InvalidDrypadArea			:= 41016,	//DrypadArea ungültig
	ERRORID_CntSpotPatternsExceeded		:= 41017,	//Anzahl SpotPatterns überschritten
	ERRORID_NoObjectAvailable			:= 41018,	//kein Object vorhanden
	ERRORID_InvalidLiquidbottle			:= 41019,	//ungültige Nummer für Flasche "Systemflüssigkeit"
	ERRORID_InvalidWastebottle			:= 41020,	//ungültige Nummer für Flasche "Waste"
	ERRORID_CntDeloDotsExceeded			:= 41021,	//Anzahl DeloDots überschritten
	ERRORID_InvalidTriggerChannel		:= 41022,	//TriggerChannel ungültig
	ERRORID_CntExposureExceeded			:= 41023,	//Anzahl Exposure überschritten
	ERRORID_CntTriplePipExceeded		:= 41024,	//Anzahl TriplePipetten überschritten
	ERRORID_CntFlipTubePinExceeded		:= 41025,	//Anzahl FlipTubePins überschritten
	ERRORID_CntLuerExceeded				:= 41026,	//Anzahl Luers überschritten
	ERRORID_CntStampExceeded			:= 41027,	//Anzahl Stempel überschritten
	ERRORID_CntNeedleExceeded			:= 41028,	//Anzahl Kanülen überschritten
	ERRORID_CntVialExceeded				:= 41029,	//Anzahl Vials überschritten
	ERRORID_CntSeptumExceeded			:= 41030,	//Anzahl Septen überschritten
	ERRORID_CntCartridgeExceeded		:= 41031,	//Anzahl Kartuschen überschritten
	ERRORID_CntPortExceeded				:= 41032,	//Anzahl Ports überschritten
	ERRORID_CntReactorExceeded			:= 41033,	//Anzahl Reaktoren überschritten
	ERRORID_Cnt4LiquidReserveExceeded	:= 41034,	//Anzahl 4LiquidReserve überschritten
	ERRORID_CntSeptumWasteExceeded		:= 41035,	//Anzahl SeptumWaste überschritten
	ERRORID_CntNeedleRackExceeded		:= 41036,	//Anzahl NeedleRacks überschritten
	ERRORID_CntSeptumRackExceeded		:= 41037,	//Anzahl SeptumRacks überschritten
	ERRORID_CntVialRackExceeded			:= 41038,	//Anzahl VialRacks überschritten
	ERRORID_CntPortRackExceeded			:= 41039,	//Anzahl PortRacks überschritten
	ERRORID_CntFlipTubeExceeded			:= 41040,	//Anzahl FlipTubes überschritten
	ERRORID_InvalidNoOfSlots			:= 41041,	//ungültiges Anzahl von Slots
	ERRORID_InvalidSlotNumber			:= 41042,	//ungultiges SlotNr
	ERRORID_InvalidNoOfSpecPoints		:= 41043,	//ungültige Anzahl von SpecPoints
	ERRORID_InvalidSpecPointNumber		:= 41044,	//ungültige SpecPointnr
	ERRORID_InvalidValveNumber			:= 41045,	//ungültige Ventilnummer
	ERRORID_InvalidHeadBoardType		:= 41046,	//
	ERRORID_HeadBoardNotAvailable		:= 41047,
	ERRORID_InvalidPumpNumber			:= 41048,
	ERRORID_CntFlipTubeRackExceeded		:= 41049,
	ERRORID_CntSpotArrayExceeded		:= 41050,	//Anzahl SpotArray überschritten
	ERRORID_InvalidHardwareRef			:= 41051,
	ERRORID_CntVacuumHandlerExceeded	:= 41052,	//Anzahl VacuumHandler überschritten
	ERRORID_InvalidRelPosZ				:= 41053,	//
	ERRORID_NoHeadCreated				:= 41054,	//kein Head angelegt, Konfiguration kann nicht aktiviert werden
	ERRORID_NoWorkplateCreated			:= 41055,	//keine Workplate angelegt, Konfiguration kann nicht aktiviert werden
	ERRORID_CntNozzleExceeded			:= 41056,	
	ERRORID_CntTwinPiezoHolderExceeded	:= 41057,	
	ERRORID_CntSinglePiezoHolderExceeded:= 41058,
	ERRORID_InvalidAxisRef				:= 41059,
	ERRORID_InvalidPiezoRef				:= 41060,
	ERRORID_InvalidNoOfRinseChannels	:= 41061,
	ERRORID_CntHighVoltTrayExceeded		:= 41062,
	ERRORID_InvalidParentObject			:= 41063,
	ERRORID_InvalidParentSlot			:= 41064,
	ERRORID_FirmwareVersionMzBase		:= 41065,
	ERRORID_CntSolenoidPipExceeded		:= 41066,
	ERRORID_CntExtruderExceeded			:= 41067,
	ERRORID_InvalidPrePeakTime			:= 41068,
	ERRORID_NoNozzleOnTool				:= 41069,
	ERRORID_InvalidExtruderSubType		:= 41070,
	ERRORID_InvalidCompressDistance		:= 41071,
	ERRORID_InvalidCompressFeed			:= 41072,
	ERRORID_InvalidExtrudeDistance		:= 41073,
	ERRORID_InvalidExtrudeFeed			:= 41074,
	ERRORID_InvalidRelaxDistance		:= 41075,
	ERRORID_InvalidRelaxFeed			:= 41076,
	ERRORID_ChangeNoOfSlotsNotAllowed	:= 41077,
	ERRORID_ChangeNoOfSpecPointsNotAllowed	:= 41078,
	ERRORID_ChangeNoOfRinseChannelsNotAllowed	:= 41079,
	ERRORID_ChangeNoOfWasteChannelsNotAllowed	:= 41080,
	ERRORID_ChangeNoOfLiquidChannelsNotAllowed	:= 41081,
	ERRORID_InvalidFactorFeed				:= 41082,
	ERRORID_InvalidFactorDistance			:= 41083,
	ERRORID_EtherCATMasterNotConfigured		:= 41084,
	ERRORID_CANopenMasterNotConfigured		:= 41085,
	ERRORID_InvalidDriveConfig				:= 41086,
	ERRORID_CntpHElectrodesExceeded			:= 41087,
	ERRORID_CntTitrationToolsExceeded		:= 41088,
	ERRORID_CntpHElectrodeCapsExceeded		:= 41089,
	ERRORID_CntpHElectrodeCapRacksExceeded 	:= 41090,
	ERRORID_InvalidAnaInputChannel		 	:= 41091,
	ERRORID_InvalidUnlockOffset		 		:= 41092,
	ERRORID_CntTwinExtruderExceeded	 		:= 41093,
	ERRORID_ExtruderInWrongSlot		 		:= 41094,
	ERRORID_UnusedExtruderSlot		 		:= 41095,
	ERRORID_CntVermesDispExceeded	 		:= 41096,
	ERRORID_CntWorkplateCameraExceeded 		:= 41097,
	ERRORID_ObjectAlreadyOnAnotherParent	:= 41098,
	ERRORID_SlotIsAlreadyOccupied			:= 41099,
	ERRORID_ObjectCanNotTakeChilds			:= 41100,
	ERRORID_ObjectNotInCollection			:= 41101,
	ERRORID_ObjectMustHaveAParent			:= 41102,
	ERRORID_ObjectHasChilds					:= 41103,
	ERRORID_InvalidDestinationSlot			:= 41104,
	ERRORID_DestinationSlotNotFree			:= 41105,
	ERRORID_CntCartridgeHolderExceeded		:= 41106,
	ERRORID_CntMultiCartridgeHolderExceeded	:= 41107,
	ERRORID_CntDummyToolExceeded			:= 41108,
	ERRORID_CntCustomUnitType1Exceeded		:= 41109,
	ERRORID_InvalidHeaterType				:= 41110,
	ERRORID_CntHybridDispenserExceeded		:= 41111,
	ERRORID_NoToolOnMasterSlot				:= 41112,
	ERRORID_CntCartridgeDispStirrerExceeded	:= 41113,
	ERRORID_InvalidPWMChannel				:= 41114,
	ERRORID_InvalidStartSpeed				:= 41115,
	ERRORID_CntCustomUnitType2Exceeded		:= 41116,
	ERRORID_CntGripperExceeded				:= 41117,
	ERRORID_CntTrayTransporterExceeded		:= 41118,
	ERRORID_CntPickPlacePipExceeded 		:= 41119,
	ERRORID_CntStackerExceeded		 		:= 41120,
	ERRORID_FDM1_NotDefined					:= 41121,
	ERRORID_FDM2_NotDefined					:= 41122,
	ERRORID_SCREWEXTR1_NotDefined			:= 41123,
	ERRORID_Stacker_NotDefined				:= 41124,
	ERRORID_InvalidNumberOfShelfes			:= 41125,
	ERRORID_PureDyne1_NotDefined			:= 41126,
	ERRORID_PureDyne2_NotDefined			:= 41127,
	ERRORID_PureDyne3_NotDefined			:= 41128
)UINT;
END_TYPE

// ---- DUTs/Enums/E_TeachTrgtOption.TcDUT
TYPE E_TeachTrgtOption :
(
	Option_PrePos := 0,
	Option_NoPrePos := 1,
	Option_AssumeInstantly := 2
)USINT;
END_TYPE

// ---- DUTs/Enums/E_TipCleaningMode.TcDUT
TYPE E_TipCleaningMode :
(
	Undefined,
    Wire,
    Brush,
    WireAndBrush	
)USINT;
END_TYPE

// ---- DUTs/Enums/E_TransferTrayCtrl.TcDUT
TYPE E_TransferTrayCtrl :
(
	LeftToSlot,
    RightToSlot,
    SlotToLeft,
	SlotToRight
)USINT;
END_TYPE

// ---- DUTs/Enums/E_TrayHollowSelection.TcDUT
{attribute 'qualified_only'}
TYPE E_TrayHollowSelection :
(
	Left,
    Centre,
    Right
)USINT;
END_TYPE

// ---- DUTs/Enums/E_TriggerOutput.TcDUT
TYPE E_TriggerOutput :
(
	PlcOutput,
	TripleTriggerModul,
	MultiZOutput,
	MultiZPWM
)USINT;
END_TYPE

// ---- DUTs/Enums/E_WashMode.TcDUT
TYPE E_WashMode :
(
	MODE_Undefiend,
	MODE_WashOutside,
	MODE_WashInside,
	MODE_WashInOutside,
	MODE_DryInside,
	MODE_DryOutside
) USINT;
END_TYPE

// ---- DUTs/ERRORID.TcDUT
TYPE ERRORID : UINT; END_TYPE

// ---- DUTs/HARDWAREGRP.TcDUT
TYPE HARDWAREGRP : UINT; END_TYPE

// ---- DUTs/Structs/ST_Action.TcDUT
{attribute 'enable_dynamic_creation'}
TYPE ST_Action :
STRUCT
	iDevice			: I_Device;
	pSequence		: POINTER TO FB_Sequence;
	eAction			: E_Action;	
	stActionData	: ST_ActionData;
	nActionId		: UINT;
	eActionStatus	: E_ActionStatus;
	eActionStatusOld: E_ActionStatus;
	nErrorId		: ERRORID;
	bExtern			: BOOL;
	nProgress		: UINT;
END_STRUCT
END_TYPE

// ---- DUTs/Structs/ST_ActionStatus.TcDUT
{attribute 'enable_dynamic_creation'}
TYPE ST_ActionStatus :
STRUCT
	nActionId	: UINT;
	eAction		: E_Action;
	nObjectId	: UINT;
	eStatus		: E_ActionStatus;
	nChannel	: USINT;
	eOldStatus	: E_ActionStatus;
END_STRUCT
END_TYPE

// ---- DUTs/Structs/ST_2DPoint.TcDUT
TYPE ST_2DPoint :
STRUCT
	X : REAL;	//X Koordinate in µm
	Y : REAL;	//X Koordinate in µm	
END_STRUCT
END_TYPE

// ---- DUTs/Structs/ST_3DDimension.TcDUT
//Größendimension von Objecten
TYPE ST_3DDimension :	
STRUCT
	Width  : REAL;	//Breite in µm
	Depth  : REAL;	//Tiefe in µm
	Height : REAL;	//Höhe in µm	
END_STRUCT
END_TYPE

// ---- DUTs/Structs/ST_3DPoint.TcDUT
TYPE ST_3DPoint :
STRUCT
	X : REAL; //X Koordinate in µm
	Y : REAL; //Y Koordinate in µm
	Z : REAL; //Z Koordinate in µm
END_STRUCT
END_TYPE

// ---- DUTs/Structs/ST_ActionData.TcDUT
TYPE ST_ActionData :
STRUCT
	eAction		: E_Action;
	nObject		: UINT;
	nTarget		: UINT;
	aParams		: ARRAY[1..19] OF DINT;
END_STRUCT
END_TYPE

// ---- DUTs/Structs/ST_ActionList.TcDUT
TYPE ST_ActionList :
STRUCT
	iDevice			: I_Device;
	pSequence		: POINTER TO FB_Sequence;
	eAction			: E_Action;	
	stActionData	: ST_ActionData;
	nActionId		: UINT;
	eActionStatus	: E_ActionStatus;
	nErrorId		: ERRORID;
	bExtern			: BOOL;
END_STRUCT
END_TYPE

// ---- DUTs/Structs/ST_AdsAdress.TcDUT
TYPE ST_AdsAdress :
STRUCT
	sNetId	: STRING(23);
	nPort	: UINT;
END_STRUCT
END_TYPE

// ---- DUTs/Structs/ST_CanMasterAddress.TcDUT
TYPE ST_CanMasterAddress :
STRUCT
	sEcMasterNetId : T_AmsNetID;
	sOwnNetId : T_AmsNetID;
	nBoxAddress : UINT; //Bezogen auf EcMaster
END_STRUCT
END_TYPE

// ---- DUTs/Structs/ST_Circle.TcDUT
TYPE ST_Circle :
STRUCT
	rX : REAL;
	rY : REAL;
	rD : REAL;
END_STRUCT
END_TYPE

// ---- DUTs/Structs/ST_EtherCATMaster.TcDUT
TYPE ST_EtherCATMaster :
STRUCT
	nDeviceId	: WORD;
	sNetId 		: T_AmsNetID;
	nCfgSlaves	: UINT;
	aStSlaveInfo : ARRAY[0..15] OF ST_EcSlaveConfigData;
END_STRUCT
END_TYPE

// ---- DUTs/Structs/ST_HardwareProcData.TcDUT
TYPE ST_HardwareProcData :
STRUCT
	nHardwareId		: DINT;		//4Byte
	nValue			: DINT;		//4Byte
	nInterpretation	: DINT;		//4Byte
END_STRUCT
END_TYPE

// ---- DUTs/Structs/ST_HardwareId.TcDUT
TYPE ST_HardwareId :
STRUCT
	nItem		: USINT;
	nParentItem : USINT;
	eGroup 		: E_HardwareGrp; 
END_STRUCT
END_TYPE

// ---- DUTs/Structs/ST_HardwareInfo.TcDUT
{attribute 'enable_dynamic_creation'}
TYPE ST_HardwareInfo :
STRUCT
	nHwId : UDINT;
	sHardwVersion : STRING(15);
	sSoftwVersion : STRING(15);
	sSoftwVersion2: STRING(3);
END_STRUCT
END_TYPE

// ---- DUTs/Structs/ST_Interaction.TcDUT
TYPE ST_Interaction :
STRUCT
	nObjectId 				: UINT;
	eInteractMessageType	: E_InteractMessageType;
	nArg1 					: DINT;
	nArg2 					: DINT;
	nArg3 					: DINT;
	nArg4 					: DINT;
END_STRUCT
END_TYPE

// ---- DUTs/Structs/ST_Line.TcDUT
TYPE ST_Line EXTENDS ST_Rectangle :
STRUCT
END_STRUCT
END_TYPE

// ---- DUTs/Structs/ST_MethResult.TcDUT
TYPE ST_MethResult :
STRUCT
	bBusy 		: BOOL;
	bCanceled	: BOOL;
	bError		: BOOL;
	nErrorId	: ERRORID;
END_STRUCT
END_TYPE

// ---- DUTs/Structs/ST_ObjHasMoved.TcDUT
TYPE ST_ObjHasMoved :
STRUCT
	ObjectId : UINT;
	DestObjId : UINT;
	DestSlotNr : UINT;
	ChangeCounter : USINT;
END_STRUCT
END_TYPE

// ---- DUTs/Structs/ST_PlcInfo.TcDUT
TYPE ST_PlcInfo :
STRUCT
	sTargetType 	: STRING(30);
	sSerialNo 		: STRING(16);
	sTwinCATBuild 	: STRING(8);
	sPlcVersion		: STRING(10);
END_STRUCT
END_TYPE

// ---- DUTs/Structs/ST_ObjectProcData.TcDUT
TYPE ST_ObjectProcData :
STRUCT
	nObjId		: DINT;
	n32Data		: ARRAY[0..13] OF DINT;
END_STRUCT
END_TYPE

// ---- DUTs/Structs/ST_Rectangle.TcDUT
TYPE ST_Rectangle :
STRUCT
	X1 : REAL;
	X2 : REAL;
	Y1 : REAL;
	Y2 : REAL;
END_STRUCT
END_TYPE

// ---- DUTs/Structs/ST_CmdData.TcDUT
//Command-Structure
//Diese Struktur wird vorrangig zum Datenaustausch zwischen GUI(Kernel) und PLC (PC_Control) benutzt
TYPE ST_CmdData :
STRUCT
	aHeader : ARRAY[0..3] OF UINT;		//8 Byte					
	n32Data	: ARRAY[0..490] OF DINT;	//491*4 Byte   1964 Byte
										//Gesamt: 1972 Byte
END_STRUCT
END_TYPE

// ---- DUTs/Structs/ST_Error.TcDUT
TYPE ST_Error :
STRUCT
	TimeStamp	: T_FILETIME;		//8Byte-Locale Systemzeit in Ticks
	//---------------------------------------------------------------------------------------
	Cmd			: UINT;				//2Byte-Kommando, welches den Fehler verursacht hat
	ObjectId	: UINT;				//2Byte-Object, welches den Fehler verursacht hat
	HardwareGrp	: HARDWAREGRP;		//2Byte-Hardwaregruppe, bei der der Fehler aufgetaucht ist
	HardwareNr	: UINT;				//2Byte-Hardwarenummer, bei der der Fehler aufgetaucht ist
	//----------------------------------------------------------------------------------------
	ErrorId		: ERRORID;			//2Byte-Fehlernummer
	POU			: E_POU;			//2Byte-Baustein, in dem der Fehler aufgetreten ist
	POUAction	: E_POUACT;			//2Byte-Methode bzw. Action, in der der Fehler aufgetreten ist
	POUState	: UINT;				//2Byte-State der Statemachine, in der der Fehler aufgetreten ist
	//----------------------------------------------------------------------------------------
	ErrorId2	: UDINT;			//4Byte-Fehlernummer2 (z.B. aus Hardware)
	MachineMode : E_MachineMode;	//1Byte-aktueller MachineMode, in dem der Fehler aufgetreten ist
	MachineState: E_MachineState;	//1Bytea-ktueller MachineState, in dem der Fehler aufgetreten ist
	//-------------------------------30 Bytes---------------------------------------------------
	//Beim ARMV7 gibt werden durch 8Byte Speicherausrichtung 32Byte belegt
END_STRUCT
END_TYPE

// ---- DUTs/Structs/ST_StepStatus.TcDUT
TYPE ST_StepStatus :
STRUCT
	nStepNr	: UINT;
	eStatus : E_StepState;
END_STRUCT
END_TYPE

// ---- DUTs/Structs/ST_WashPoint.TcDUT
TYPE ST_WashPoint EXTENDS ST_3DPoint :
STRUCT
	nRinseChannel : USINT;
END_STRUCT
END_TYPE

// ---- DUTs/Structs/ST_WashStep.TcDUT
TYPE ST_WashStep :
STRUCT
	eMode : E_WashMode;
	nParam1 : DINT;
	nParam2 : DINT;
	nParam3 : DINT;
	nParam4 : DINT;
END_STRUCT
END_TYPE

// ---- DUTs/Structs/ST_WasteChannel.TcDUT
TYPE ST_WasteChannel :
STRUCT
	nNr		 	: USINT;
	nSpecPointNr: USINT;
	nPumpNr	 	: USINT;
	nBottleNr	: USINT;
END_STRUCT
END_TYPE

// ---- DUTs/Structs/ST_LiquidChannel.TcDUT
TYPE ST_LiquidChannel :
STRUCT
	nNr		 : USINT;
	nSlotNr	 : USINT;
	nWasteCh : USINT;
	nBottleNr: USINT;
	pGearPump: POINTER TO FB_GearPump;
END_STRUCT
END_TYPE

// ---- DUTs/Structs/ST_RinseChannel.TcDUT
TYPE ST_RinseChannel :
STRUCT
	nPumpNr	 	: USINT;
	nValveNr	: USINT;
	nStartSpeed	: USINT;
	nRatedSpeed : USINT;
	nStartTime	: UINT;
END_STRUCT
END_TYPE

// ---- DUTs/Unions/U_AdsData.TcDUT
TYPE U_AdsData :
UNION
	stCmdData	: ST_CmdData;
	aUINT_1000	: ARRAY[0..999] OF UINT;
	aDINT_20	: ARRAY[0..19] OF DINT;
	aDINT_40	: ARRAY[0..39] OF DINT;
	ConfigId	: GUID;
END_UNION
END_TYPE

// ---- DUTs/Unions/U_ByteArr4_DINT.TcDUT
TYPE U_ByteArr4_DINT :
UNION
	aBytes : ARRAY[0..3] OF BYTE;
	nDINT  : DINT;
END_UNION
END_TYPE

// ---- DUTs/Unions/U_SDO_DATA.TcDUT
TYPE U_SDO_DATA :
UNION
	aData : ARRAY[0..3] OF BYTE;
	nData : DINT;
	sData : STRING(20);
END_UNION
END_TYPE

// ---- FirmwUpdate/E_FirmwUpdState.TcDUT
TYPE E_FirmwUpdState :
(
	LoadFile,
	Connect,
	GetStatus,
	ProgramStart,
	SetMTA,
	ProgramClear,
	Programming,
	WaitForBootup,
	Ready,
	Error
);
END_TYPE

// ---- FirmwUpdate/E_S19RecordState.TcDUT
TYPE E_S19RecordState :
(
	Undefined := 0,
	Valid,
	BlockEnd,
	NotComplete,
	CRC_Error,
	Line_Error
)USINT;
END_TYPE

// ---- FirmwUpdate/ST_FirmwUpdInfo.TcDUT
TYPE ST_FirmwUpdInfo :
STRUCT
	nBytesToWrite 	: UDINT;
	nWrittenBytes	: UDINT;
	eActState 		: E_FirmwUpdState;	
END_STRUCT
END_TYPE

// ---- GCode/E_SAF_State.TcDUT
TYPE E_SAF_State :
(
	Control := 2,
	Run := 3
)UDINT;
END_TYPE

// ---- GCode/ST_GCodeInfo2.TcDUT
TYPE ST_GCodeInfo2 :
STRUCT
		nTargetObjId	: UINT;
END_STRUCT
END_TYPE

// ---- GCode/ST_GCodeRef.TcDUT
TYPE ST_GCodeRef :
STRUCT
	sNciToPlc	     AT %I* : NCTOPLC_NCICHANNEL_REF;
	sPlcToNci	     AT %Q* : PLCTONC_NCICHANNEL_REF;
	aToolTable		: ARRAY[1..GCode.cMaxGCodeTools] OF ST_GCodeTool;
	aTargetTable	: ARRAY[1..GCode.cMaxGCodeTargets] OF UINT; //ObjectIDs ausgewählten Targets
	pCurrentTool	: POINTER TO FB_GCodeTool;
	pHead			: POINTER TO FB_MzHead;
	pWaitPoint		: POINTER TO FB_TargetBase;		
	sZeroShiftDesc	: Tc2_NCI.ZeroShiftDesc;
	lrNcOverride 	: LREAL := 100.0;
	stStartPos		: ST_3DPoint;
	fbLimitCuboid	: FB_Cuboid;
	aSequenceIds	: ARRAY[1..5] OF UDINT;
END_STRUCT
END_TYPE

// ---- GCode/ST_GCodeTool.TcDUT
TYPE ST_GCodeTool :
STRUCT
	bIsUsed			: BOOL;	//wird durch AssignRParams gesetzt
	pMzTool			: POINTER TO FB_GCodeTool;
	bIsInAction1	: BOOL;	//True, wenn in Pause gegangen wird und gerade mit Action1 geprintet wird
	bIsInAction2 	: BOOL;	//True, wenn in Pause gegangen wird und gerade mit Action2 geprintet wird
	bIsInAction3 	: BOOL;	//True, wenn in Pause gegangen wird und gerade mit Action3 geprintet wird
	tDelayStart 	: TIME;	//Startverzögerung nach Continue
END_STRUCT
END_TYPE

// ---- GCode/ST_NciInfo.TcDUT
TYPE ST_NciInfo :
STRUCT
	Mode : UDINT;
	FileOffset : UDINT;
	FileName : ARRAY[1..260] OF USINT;
END_STRUCT
END_TYPE

// ---- GCode/ST_GCodeInfo.TcDUT
TYPE ST_GCodeInfo :
STRUCT
	nNciState	: UDINT;
	nFileNr		: UDINT;
	nFileOffset : UDINT;
	nCurrentObj	: UINT;
	eGCodeState : E_GCodeState;
END_STRUCT
END_TYPE

// ---- Hardware/EL70xxDrive/E_EL70xx_EncoderType.TcDUT
{attribute 'qualified_only'}
TYPE E_EL70xx_EncoderType :
(
	InternEncoder := 0,
	InternCounter := 1,
	ExternSingleturnAbs := 2
) USINT;
END_TYPE

// ---- Hardware/EL70xxDrive/E_EL70xx_StartType.TcDUT
{attribute 'qualified_only'}
TYPE E_EL70xx_StartType :
(
	Absolute := 16#0001,
	Relative := 16#0002,
	EndlessPlus := 16#0003,
	EndlessMinus := 16#0004,
	CaliPlcCam := 16#6000,
	CaliHwSync := 16#6100,
	SetCalibration := 16#6E00,
	ClearCalibration := 16#6F00
)UINT;
END_TYPE

// ---- Hardware/EL70xxDrive/ST_EL70xx_POS_Control.TcDUT
TYPE ST_EL70xx_POS_Control :
STRUCT
	Execute 		AT %Q* : BIT;
	EmergencyStop 	AT %Q* : BIT;
	TargetPosition	AT %Q* : DINT;
	Velocity		AT %Q* : INT;
	StartType		AT %Q* : E_EL70xx_StartType;
	Acceleration	AT %Q* : UINT;
	Deceleration	AT %Q* : UINT;
END_STRUCT
END_TYPE

// ---- Hardware/EL70xxDrive/ST_EL70xx_POS_Status.TcDUT
TYPE ST_EL70xx_POS_Status :
STRUCT
	Busy  			AT%I* : BIT;
	InTarget  		AT%I* : BIT;
	Warning  		AT%I* : BIT;
	Error 			AT%I* : BIT;
	Calibrated  	AT%I* : BIT;
	//ReadyToExecute  AT%I* : BIT;
	ActualPosition  AT%I* : DINT;
END_STRUCT
END_TYPE

// ---- Hardware/EL70xxDrive/ST_EL70xx_STM_Control.TcDUT
TYPE ST_EL70xx_STM_Control :
STRUCT
	Enable			AT %Q* : BIT;
	Reset			AT %Q* : BIT;
	ReduceTorque 	AT %Q* : BIT;	//Spulenstrom reduzieren
END_STRUCT
END_TYPE

// ---- Hardware/EL70xxDrive/ST_EL70xx_STM_Status.TcDUT
TYPE ST_EL70xx_STM_Status :
STRUCT
	ReadyToEnable 	AT %I* : BIT;
	Ready 			AT %I* : BIT;
	Warning 		AT %I* : BIT;
	Error  			AT %I* : BIT;
END_STRUCT
END_TYPE

// ---- Hardware/E_CoDS402HomingState.TcDUT
TYPE E_CoDS402HomingState :
(
	HomingInProgress,
	HomingInteruptedOrNotReached,
	HomingAttainedButNotReached,
	HomingSuccess,
	HomingError
);
END_TYPE

// ---- Hardware/HuberUnistat/E_UnistatState.TcDUT
TYPE E_UnistatState :
(
	Error := -1,
	Off := 0,
	On := 1
)DINT;
END_TYPE

// ---- Hardware/HuberUnistat/E_Unitstat_Command.TcDUT
{attribute 'qualified_only'}
{attribute 'strict'}
TYPE E_Unitstat_Command :
(
	Get_TempActualIntern,
	Get_TempActualExtern,
	Get_TempSetPoint,
	Get_Status,
	Set_TempSetPoint,
	Start_TempControl,
	Stop_TempControl
)USINT;
END_TYPE

// ---- Hardware/IOExpander/ST_PulseTrainChannel.TcDUT
TYPE ST_PulseTrainChannel :
STRUCT
	nPeriod AT %Q* : UINT;
	nPulse AT %Q* : UINT;
	nNoOfPulses AT %Q* : UINT;
	nCtrl AT %Q* : USINT;
	nEnabled AT %Q* : USINT := 1;
	nState AT %I* : USINT;
END_STRUCT
END_TYPE

// ---- Hardware/MultiZ/Heater/E_MzHeaterType.TcDUT
TYPE E_MzHeaterType :
(
	Nothing,
	SingleHeater,	//MB
	TwinHeater,		//HT-Heater
	HeaterCooler	//Heizer und Kühler
);
END_TYPE

// ---- Hardware/Safety/E_SafetyCtrl.TcDUT
{attribute 'qualified_only'}
TYPE E_SafetyCtrl :
(
	Unlock,
	Lock,
	Quit
);
END_TYPE

// ---- Hardware/Safety/E_SafetyState.TcDUT
{attribute 'qualified_only'}
{attribute 'strict'}
TYPE E_SafetyState :
(
	Init,
	Unlocked,
	Locked,
	UnlockedBoxCtcOpen,
	UnlockedBoxCtcClosed,
	EmergencyStopPressed,
	EmergencyStopReleased,
	Error
)USINT;
END_TYPE

// ---- Hardware/E_CoDS402States.TcDUT
TYPE E_CoDS402States :
(
	DS402STATE_Notspecified := 0,
	DS402STATE_NotReadyToSwitchOn,
	DS402STATE_SwitchOnDisabled,
	DS402STATE_ReadyToSwitchOn,
	DS402STATE_SwitchedOn,
	DS402STATE_OperationEnabled,
	DS402STATE_QuickStopActive,
	DS402STATE_FaultReactionActive,
	DS402STATE_HomingInProgess,
	DS402STATE_HomingCompleted,
	DS402STATE_Fault
)UINT;
END_TYPE

// ---- Hardware/LiquidReserve/E_TMCMCommand.TcDUT
TYPE E_TMCMCommand :
(
	//Commands setzt sich aus TMCL-Instruction + TMCL-Type zusammen
	ROTATE_R := 256,			//MSB= ROR=1 , LSB= 0
	ROTATE_L := 512,			//MSB= ROL=2 , LSB= 0
	STOP := 768,				//MSB= STOP=3 , LSB=0
	MOVE_ABS := 1024,			//MSB= MVP=4 , LSB= ABS= 0
	MOVE_REL := 1025,			//MSB= MVP=4 , LSB= REL= 1
	SET_SPEED := 1284,			//MSB= SAP=5 , LSB= max positioning speed= 4
	GET_ACT_SPEED := 1539,		//MSB= GAP=6 , LSB= actual speed= 3
	GET_POS_REACHED := 1544		//MSB= GAP=6 , LSB= position reached= 8
)UINT;
END_TYPE

// ---- Hardware/MultiZ/E_MzToolType.TcDUT
TYPE E_MzToolType :
(
	TOOL_TYPE_None := 0,
	TOOL_TYPE_Cartridge := 1,
	TOOL_TYPE_PiezoPip := 2,
	TOOL_TYPE_Stamp := 3,
	TOOL_TYPE_TipEjector := 4,
	TOOL_TYPE_PowderPip := 5,
	TOOL_TYPE_HTExtruder := 6,
	TOOL_TYPE_PiezoMaster := 7,
	TOOL_TYPE_PiezoSlave := 8,
	TOOL_TYPE_PiezoSingle := 9,
	TOOL_TYPE_SyringeExtruder := 10,
	TOOL_TYPE_CoolingCartridge := 11,
	TOOL_TYPE_HTCartrigde := 12,
	TOOL_TYPE_PowderPipGen2 := 13,
	TOOL_TYPE_Gripper :=14,
	TOOL_TYPE_GenericPEXTool:= 254	//PEX = Portexpander
)USINT;
END_TYPE

// ---- Hardware/MultiZ/GPIO/E_GPInputMode.TcDUT
TYPE E_GPInputMode :
(
	Disabled,
	Analog,
	Digital,
	Limits
);
END_TYPE

// ---- Hardware/MultiZ/Piezo/E_DispenserMode.TcDUT
TYPE E_DispenserMode :
(
	MODE_None,
	MODE_Piezo,
	MODE_Solenoid
)USINT;
END_TYPE

// ---- Hardware/MultiZ/ST_CANopenObject.TcDUT
TYPE ST_CANopenObject :
STRUCT
	nIndex 		: DWORD;
	nSubIndex 	: DWORD;
	nLength 	: DWORD;
END_STRUCT
END_TYPE

// ---- Hardware/MultiZ/ST_StampSupport.TcDUT
TYPE ST_StampSupport :
STRUCT
	bAngleReached 		AT %I* : BOOL; //PDO (Bit0 StampState)
	bLocked				AT %I* : BOOL; //PDO (Bit1 StampState)
	bInitSpinOk			AT %I* : BOOL; //PDO (Bit2 StampState)
	bInitLockOk			AT %I* : BOOL; //PDO (Bit3 StampState)
	bError				AT %I* : BOOL; //PDO (Bit4 StampState)
	bStampInMagazine 	AT %I* : BOOL; //PDO (Bit5 StampState)
	bStampInSupport 	AT %I* : BOOL; //PDO (Bit6 StampState)
	
	bCtrl			: BOOL;		//SDO(RW)
	nMode			: USINT;	//SDO(RW)
	nAngleSetpoint	: INT;		//SDO(RW)
	nAngleMax		: INT;		//SDO(RO)
	nSpinSpeed		: UDINT; 	//SDO(RW)
	bLock			: BOOL;		//SDO(RW)
	nUnlockOffset	: DINT;		//SDO(RW)
	bLight			: BOOL;		//SDO(RW)
END_STRUCT
END_TYPE

// ---- Hardware/MultiZ/ST_StrobTrigger.TcDUT
TYPE ST_StrobTrigger :
STRUCT
	//aDroplist muss an erster Stelle stehen, da bei ARM7 die 4Byte Speicherausrichtung
	//Probleme bei der weiteren Verarbeitung macht
	aDroplist	: ARRAY[1..16] OF USINT;
	bTest		: BOOL;
	nCamDelay 	: UINT;
	nStrobDelay : UINT;
	nStrobDelay2 : UINT;
	bDroplistActive : BOOL;
END_STRUCT
END_TYPE

// ---- Hardware/MultiZ/ST_ZAxisRef_In.TcDUT
TYPE ST_ZAxisRef_In :
STRUCT
	nStatus		AT %I* : USINT;
	nCurrentPos AT %I* : DINT;
	nToolState	AT %I* : USINT;
	nError		AT %I* : USINT;
END_STRUCT
END_TYPE

// ---- Hardware/MultiZ/ST_ZAxisRef_Out.TcDUT
TYPE ST_ZAxisRef_Out :
STRUCT
	nCtrl			AT %Q* : USINT;	//PDO
	nMode			AT %Q* : USINT;	//PDO
	nTrgtPos		AT %Q* : DINT;	//PDO
	nVelo			AT %Q* : DINT;	//PDO
	nToolCtrl		AT %Q* : BYTE;	//PDO
	nForceThrshld	: UINT;			//SDO
	nForcePos		: DINT;			//SDO
	nForceVelo		: UINT;			//SDO
	bTipEjectExist	: BOOL;			//SDO
	
	nToolEnable		: USINT;		//Sdo
END_STRUCT
END_TYPE

// ---- Hardware/MultiZ/ST_ZAxisStatus.TcDUT
TYPE ST_ZAxisStatus :
STRUCT
	bError			: BOOL;	//Achse ist in Fehler
	bCmdAborted 	: BOOL;	//Achse wurde gestoppt
	bHasJob			: BOOL;	//Achse hat einen Fahrauftrag
	bIsMoving		: BOOL;	//Achse ist gerade in Bewegung
	bIsHoming		: BOOL;	//Achse wird gerade referenziert
	bIsHomed		: BOOL;	//Achse ist referenziert
	nADSError		: UINT;	
END_STRUCT
END_TYPE

// ---- Hardware/MultiZ/ST_ZGPIO_AnaIn.TcDUT
TYPE ST_ZGPIO_AnaIn :
STRUCT
	nValue		AT %I* : INT;	//Pdo
	nTrigger	: USINT;		//Sdo
	nLimit		: INT;			//Sdo
	nDelta		: INT;			//Sdo
END_STRUCT
END_TYPE

// ---- Hardware/MultiZ/ST_ZGPIO_PWM_ANA.TcDUT
TYPE ST_ZGPIO_PWM_ANA :
STRUCT
	bEnable	: BOOL;	//wird per SDO gesetzt
	nValue	: UINT;		//wird per SDO gesetzt
END_STRUCT
END_TYPE

// ---- Hardware/MultiZ/ST_ZSensorCalibration.TcDUT
TYPE ST_ZSensorCalibration :
STRUCT
	nId : DINT;
	nAxis : USINT;
	rValue : REAL;
END_STRUCT
END_TYPE

// ---- Hardware/PTOStepper/ST_PTOStepperRef.TcDUT
TYPE ST_PTOStepperRef :
STRUCT
	nCounterValue 		AT %I* : UINT;
	bCounterUnderflow	AT %I* : BOOL;
	bCounterOverflow	AT %I* : BOOL;
	bSetCounter			AT %Q* : BOOL;
	nFrequencyValue 	AT %Q* : UINT;
	nSetCounterValue	AT %Q* : UINT;
END_STRUCT
END_TYPE

// ---- Hardware/Reactor/E_ReactDrive.TcDUT
TYPE E_ReactDrive :
(
	Clamp := 1,
	CoverHoriz := 2,
	CoverVerti := 3,
	CoverBoth := 4,
	Complete
)USINT;
END_TYPE

// ---- Hardware/ST_CANInterfaceBuffer.TcDUT
TYPE ST_CANInterfaceBuffer :
STRUCT
	hList	: T_HLINKEDLIST;
	aNodes  : ARRAY[0..5] OF T_LinkedListEntry;
	bExecute: BOOL;
	bBusy	: BOOL;
	bError	: BOOL;
	nTxIdent: UINT;
	nTxDlc	: USINT;
	aTxData	: ARRAY[0..7] OF USINT;
	nRxIdent: UINT;
	nRxDlc	: USINT;
	aRxData	: ARRAY[0..7] OF USINT;	
END_STRUCT
END_TYPE

// ---- Hardware/TipCalibrator/ST_TipCalibrator.TcDUT
TYPE ST_TipCalibrator :
STRUCT
	bXSensor AT %I* : BOOL;
	bYSensor AT %I* : BOOL;
	bInvert	 : BOOL; //für Linmotantriebe	
END_STRUCT
END_TYPE

// ---- Hardware/TipCleaner/ST_TipCleanerRef.TcDUT
TYPE ST_TipCleanerRef :
STRUCT
	stAdsAdress			: ST_AdsAdress;
	//Eingänge
	nStatus		 		AT %I* : UINT;	//Statusword 
	nModeDisp			AT %I* : USINT; //Aktueller Wert von Mode of Operation
	nCurrentPos			AT %I* : DINT;	//Aktuelle Position
	//bOpticSensor		AT %I* : BOOL;	//Lichtschranke Digitaler Eingang 0

	//Ausgänge
	nControl			AT %Q* : UINT; 	//Controlword
	nMode				AT %Q* : USINT;	//Mode of Operations
	nTargetPos			AT %Q* : DINT;	//Target Position 
	bVDD5V				AT %Q* : BOOL;	//Digitaler Ausgang1 5V VDD
 END_STRUCT
END_TYPE

// ---- Hardware/TMCM-1140/E_TMCM_HomingMethode.TcDUT
TYPE E_TMCM_HomingMethode :
(
	NoHoming := 0,
	SearchLeftEndSwitchNextIndex := 1,
	SearchRightEndSwitchNextIndex := 2,
	SearchPosHomeSwitchNextIndex := 3,
	SearchNegHomeSwitchNextIndex := 5,
	SearchLeftEndSwitch := 17,
	SearchRightEndSwitch := 18,
	SearchPosHomeSwitch := 19,
	SearchNegHomeSwitch := 21,
	SearchNextIndexInNegDir := 33,
	SearchNextIndesInPosDir := 35,
	ActualPosAsHomePos := 36
)USINT;
END_TYPE

// ---- Hardware/TMCM-1140/E_TMCM_SwitchConfig.TcDUT
TYPE E_TMCM_SwitchConfig :
(
	Activated := 0, 
	Deactivated := 1,
	Inverted := 2
);
END_TYPE

// ---- Hardware/TMCM-1140/E_TMCM_VeloDim.TcDUT
{attribute 'qualified_only'}
{attribute 'strict'}
TYPE E_TMCM_VeloDim :
(
	INTERN := 0,
	RPM := 164,
	PPS := 181
)USINT;
END_TYPE

// ---- Hardware/XYDrive/E_XYOrientation.TcDUT
{attribute 'qualified_only'}
{attribute 'strict'}
TYPE E_XYOrientation :
(
	X,
	Y
)USINT;
END_TYPE

// ---- Objects/ST_Shelf.TcDUT
TYPE ST_Shelf :
STRUCT
	nPosition 	: DINT;
	bConfigured : BOOL;
END_STRUCT
END_TYPE

// ---- Objects/ST_POINTER2.TcDUT
{attribute 'enable_dynamic_creation'}
TYPE ST_POINTER2 :
STRUCT
	pContent:  PVOID;
	pPrev	:  PVOID;
	pNext	:  PVOID;	
END_STRUCT
END_TYPE

// ---- Sequence/E_SequenceState.TcDUT
TYPE E_SequenceState :
(
	State_Idle,
	State_Start,
	State_Active,
	State_PauseRequest,
	State_Pause,
	State_Continue,
	State_Cancel,
	State_Canceled,
	State_Ready,
	State_Error
)USINT;
END_TYPE

// ---- Sequence/E_StepState.TcDUT
TYPE E_StepState :
(
	STEPSTATUS_Idle := 0,
	STEPSTATUS_InQueue,
	STEPSTATUS_Active,
	STEPSTATUS_Pause,
	STEPSTATUS_Ready,
	STEPSTATUS_Error
)USINT;
END_TYPE

// ---- Sequence/ST_Pointer.TcDUT
{attribute 'enable_dynamic_creation'}
TYPE ST_Pointer :
STRUCT
	pContent:  POINTER TO PVOID;
	pPrev	:  POINTER TO PVOID;
	pNext	:  POINTER TO PVOID;
END_STRUCT
END_TYPE

